LIN {X 0,Y 312.863,Z 418.471,A -85,B 0,C 180,E1 -15890.336,E2 -15890.336} C_VEL
LIN {X 0,Y 316.327,Z 432.665,A -85,B 0,C 180,E1 -15893.379,E2 -15893.379} C_VEL
LIN {X 0,Y 317.208,Z 437.346,A -85,B 0,C 180,E1 -15894.325,E2 -15894.325} C_VEL
LIN {X 0,Y 317.095,Z 438.182,A -85,B 0,C 180,E1 -15894.467,E2 -15894.467} C_VEL
LIN {X 0,Y 321.932,Z 475.252,A -85,B 0,C 180,E1 -15895.925,E2 -15895.925} C_VEL
LIN {X 0,Y 326.168,Z 512.092,A -85,B 0,C 180,E1 -15897.258,E2 -15897.258} C_VEL
LIN {X 0,Y 323.203,Z 607.757,A -85,B 0,C 180,E1 -15899.36,E2 -15899.36} C_VEL
LIN {X 0,Y 322.103,Z 623.409,A -85,B 0,C 180,E1 -15899.924,E2 -15899.924} C_VEL
LIN {X 0,Y 320.466,Z 638.482,A -85,B 0,C 180,E1 -15900.704,E2 -15900.704} C_VEL
LIN {X 0,Y 318.45,Z 652.595,A -85,B 0,C 180,E1 -15901.674,E2 -15901.674} C_VEL
LIN {X 0,Y 316.125,Z 666.999,A -85,B 0,C 180,E1 -15902.948,E2 -15902.948} C_VEL
LIN {X 0,Y 313.926,Z 680.599,A -85,B 0,C 180,E1 -15904.472,E2 -15904.472} C_VEL
LIN {X 0,Y 311.576,Z 693.378,A -85,B 0,C 180,E1 -15906.222,E2 -15906.222} C_VEL
LIN {X 0,Y 309.65,Z 704.13,A -85,B 0,C 180,E1 -15908.007,E2 -15908.007} C_VEL
LIN {X 0,Y 307.924,Z 714.131,A -85,B 0,C 180,E1 -15909.979,E2 -15909.979} C_VEL
LIN {X 0,Y 306.386,Z 723.981,A -85,B 0,C 180,E1 -15912.306,E2 -15912.306} C_VEL
LIN {X 0,Y 305.308,Z 732.423,A -85,B 0,C 180,E1 -15914.718,E2 -15914.718} C_VEL
LIN {X 0,Y 304.657,Z 739.918,A -85,B 0,C 180,E1 -15917.341,E2 -15917.341} C_VEL
LIN {X 0,Y 304.529,Z 746.052,A -85,B 0,C 180,E1 -15920.032,E2 -15920.032} C_VEL
LIN {X 0,Y 304.716,Z 750.636,A -85,B 0,C 180,E1 -15922.635,E2 -15922.635} C_VEL
LIN {X 0,Y 304.965,Z 753.357,A -85,B 0,C 180,E1 -15924.711,E2 -15924.711} C_VEL
LIN {X 0,Y 305.159,Z 755.666,A -85,B 0,C 180,E1 -15927.36,E2 -15927.36} C_VEL
LIN {X 0,Y 305.45,Z 756.378,A -85,B 0,C 180,E1 -15928.681,E2 -15928.681} C_VEL
LIN {X 0,Y 305.657,Z 756.769,A -85,B 0,C 180,E1 -15929.999,E2 -15929.999} C_VEL
LIN {X 0,Y 305.424,Z 756.792,A -85,B 0,C 180,E1 -15931.318,E2 -15931.318} C_VEL
LIN {X 0,Y 304.976,Z 755.908,A -85,B 0,C 180,E1 -15933.964,E2 -15933.964} C_VEL
LIN {X 0,Y 304.626,Z 753.778,A -85,B 0,C 180,E1 -15936.623,E2 -15936.623} C_VEL
LIN {X 0,Y 304.345,Z 750.421,A -85,B 0,C 180,E1 -15939.302,E2 -15939.302} C_VEL
LIN {X 0,Y 304.424,Z 745.812,A -85,B 0,C 180,E1 -15941.991,E2 -15941.991} C_VEL
LIN {X 0,Y 305.049,Z 739.867,A -85,B 0,C 180,E1 -15944.68,E2 -15944.68} C_VEL
LIN {X 0,Y 306.24,Z 732.446,A -85,B 0,C 180,E1 -15947.357,E2 -15947.357} C_VEL
LIN {X 0,Y 307.878,Z 724.631,A -85,B 0,C 180,E1 -15949.675,E2 -15949.675} C_VEL
LIN {X 0,Y 309.953,Z 715.588,A -85,B 0,C 180,E1 -15951.899,E2 -15951.899} C_VEL
LIN {X 0,Y 312.669,Z 704.202,A -85,B 0,C 180,E1 -15954.217,E2 -15954.217} C_VEL
LIN {X 0,Y 315.71,Z 691.846,A -85,B 0,C 180,E1 -15956.258,E2 -15956.258} C_VEL
LIN {X 0,Y 318.808,Z 679.206,A -85,B 0,C 180,E1 -15957.952,E2 -15957.952} C_VEL
LIN {X 0,Y 321.789,Z 665.625,A -85,B 0,C 180,E1 -15959.432,E2 -15959.432} C_VEL
LIN {X 0,Y 324.584,Z 652.223,A -85,B 0,C 180,E1 -15960.584,E2 -15960.584} C_VEL
LIN {X 0,Y 327.156,Z 637.542,A -85,B 0,C 180,E1 -15961.574,E2 -15961.574} C_VEL
LIN {X 0,Y 329.294,Z 622.301,A -85,B 0,C 180,E1 -15962.336,E2 -15962.336} C_VEL
LIN {X 0,Y 330.686,Z 606.3,A -85,B 0,C 180,E1 -15962.905,E2 -15962.905} C_VEL
LIN {X 0,Y 332.705,Z 555.604,A -85,B 0,C 180,E1 -15964.025,E2 -15964.025} C_VEL
LIN {X 0,Y 334.221,Z 512.744,A -85,B 0,C 180,E1 -15964.965,E2 -15964.965} C_VEL
LIN {X 0,Y 331.794,Z 490.509,A -85,B 0,C 180,E1 -15965.887,E2 -15965.887} C_VEL
LIN {X 0,Y 327.9,Z 463.19,A -85,B 0,C 180,E1 -15967.187,E2 -15967.187} C_VEL
LIN {X 0,Y 325.208,Z 447.828,A -85,B 0,C 180,E1 -15968.019,E2 -15968.019} C_VEL
LIN {X 0,Y 320.37,Z 437.85,A -85,B 0,C 180,E1 -15969.057,E2 -15969.057} C_VEL
LIN {X 0,Y 318.662,Z 434.062,A -85,B 0,C 180,E1 -15969.474,E2 -15969.474} C_VEL
LIN {X 0,Y 315.48,Z 422.569,A -85,B 0,C 180,E1 -15972.365,E2 -15972.365} C_VEL
LIN {X 0,Y 312.299,Z 412.488,A -85,B 0,C 180,E1 -15975.122,E2 -15975.122} C_VEL
LIN {X 0,Y 308.681,Z 402.063,A -85,B 0,C 180,E1 -15978.244,E2 -15978.244} C_VEL
LIN {X 0,Y 305.398,Z 393.062,A -85,B 0,C 180,E1 -15981.242,E2 -15981.242} C_VEL
LIN {X 0,Y 305.451,Z 393.062,A -85,B 0,C 180,E1 -15984.886,E2 -15984.886} C_VEL
LIN {X 0,Y 305.432,Z 393.066,A -85,B 0,C 180,E1 -15988.358,E2 -15988.358} C_VEL
LIN {X 0,Y 305.464,Z 393.064,A -85,B 0,C 180,E1 -15991.108,E2 -15991.108} C_VEL
LIN {X 0,Y 305.467,Z 393.064,A -85,B 0,C 180,E1 -15994.079,E2 -15994.079} C_VEL
LIN {X 0,Y 305.443,Z 393.06,A -85,B 0,C 180,E1 -15998.399,E2 -15998.399} C_VEL
LIN {X 0,Y 305.486,Z 393.06,A -85,B 0,C 180,E1 -16001.211,E2 -16001.211} C_VEL
LIN {X 0,Y 305.557,Z 393.047,A -85,B 0,C 180,E1 -16005.345,E2 -16005.345} C_VEL
LIN {X 0,Y 305.611,Z 393.035,A -85,B 0,C 180,E1 -16009.399,E2 -16009.399} C_VEL
LIN {X 0,Y 305.733,Z 393.029,A -85,B 0,C 180,E1 -16012.073,E2 -16012.073} C_VEL
LIN {X 0,Y 305.647,Z 393.034,A -85,B 0,C 180,E1 -16014.723,E2 -16014.723} C_VEL
LIN {X 0,Y 305.923,Z 393,A -85,B 0,C 180,E1 -16018.684,E2 -16018.684} C_VEL
LIN {X 0,Y 305.936,Z 392.992,A -85,B 0,C 180,E1 -16021.317,E2 -16021.317} C_VEL
LIN {X 0,Y 305.776,Z 392.982,A -85,B 0,C 180,E1 -16026.648,E2 -16026.648} C_VEL
LIN {X 0,Y 305.674,Z 393.019,A -85,B 0,C 180,E1 -16029.262,E2 -16029.262} C_VEL
LIN {X 0,Y 305.574,Z 393.019,A -85,B 0,C 180,E1 -16033.297,E2 -16033.297} C_VEL
LIN {X 0,Y 305.542,Z 393.033,A -85,B 0,C 180,E1 -16036.023,E2 -16036.023} C_VEL
LIN {X 0,Y 305.532,Z 393.035,A -85,B 0,C 180,E1 -16039.427,E2 -16039.427} C_VEL
LIN {X 0,Y 305.447,Z 393.055,A -85,B 0,C 180,E1 -16043.027,E2 -16043.027} C_VEL
LIN {X 0,Y 305.442,Z 393.042,A -85,B 0,C 180,E1 -16046.191,E2 -16046.191} C_VEL
LIN {X 0,Y 305.438,Z 393.064,A -85,B 0,C 180,E1 -16049.034,E2 -16049.034} C_VEL
LIN {X 0,Y 305.428,Z 393.046,A -85,B 0,C 180,E1 -16051.954,E2 -16051.954} C_VEL
LIN {X 0,Y 305.454,Z 393.062,A -85,B 0,C 180,E1 -16055.115,E2 -16055.115} C_VEL
LIN {X 0,Y 305.445,Z 393.061,A -85,B 0,C 180,E1 -16059.257,E2 -16059.257} C_VEL
LIN {X 0,Y 305.406,Z 393.058,A -85,B 0,C 180,E1 -16059.929,E2 -16059.929} C_VEL
LIN {X 0,Y 306.44,Z 395.935,A -85,B 0,C 180,E1 -16060.224,E2 -16060.224} C_VEL
LIN {X 0,Y 308.625,Z 398.473,A -85,B 0,C 180,E1 -16060.717,E2 -16060.717} C_VEL
LIN {X 0,Y 310.885,Z 401.914,A -85,B 0,C 180,E1 -16061.24,E2 -16061.24} C_VEL
LIN {X 0,Y 317.694,Z 411.904,A -85,B 0,C 180,E1 -16062.735,E2 -16062.735} C_VEL
LIN {X 0,Y 325.78,Z 424.373,A -85,B 0,C 180,E1 -16064.399,E2 -16064.399} C_VEL
LIN {X 0,Y 335.544,Z 441.537,A -85,B 0,C 180,E1 -16066.307,E2 -16066.307} C_VEL
LIN {X 0,Y 336.591,Z 443.642,A -85,B 0,C 180,E1 -16066.508,E2 -16066.508} C_VEL
LIN {X 0,Y 334.079,Z 511.752,A -85,B 0,C 180,E1 -16067.994,E2 -16067.994} C_VEL
LIN {X 0,Y 333.569,Z 531.567,A -85,B 0,C 180,E1 -16068.547,E2 -16068.547} C_VEL
LIN {X 0,Y 332.676,Z 546.26,A -85,B 0,C 180,E1 -16069.186,E2 -16069.186} C_VEL
LIN {X 0,Y 331.305,Z 560.291,A -85,B 0,C 180,E1 -16070.013,E2 -16070.013} C_VEL
LIN {X 0,Y 329.701,Z 573.58,A -85,B 0,C 180,E1 -16071.038,E2 -16071.038} C_VEL
LIN {X 0,Y 327.599,Z 586.902,A -85,B 0,C 180,E1 -16072.311,E2 -16072.311} C_VEL
LIN {X 0,Y 325.278,Z 599.133,A -85,B 0,C 180,E1 -16073.74,E2 -16073.74} C_VEL
LIN {X 0,Y 322.637,Z 611.425,A -85,B 0,C 180,E1 -16075.505,E2 -16075.505} C_VEL
LIN {X 0,Y 319.968,Z 622.521,A -85,B 0,C 180,E1 -16077.445,E2 -16077.445} C_VEL
LIN {X 0,Y 317.476,Z 631.8,A -85,B 0,C 180,E1 -16079.394,E2 -16079.394} C_VEL
LIN {X 0,Y 314.87,Z 640.813,A -85,B 0,C 180,E1 -16081.687,E2 -16081.687} C_VEL
LIN {X 0,Y 312.617,Z 648.371,A -85,B 0,C 180,E1 -16084.06,E2 -16084.06} C_VEL
LIN {X 0,Y 310.556,Z 655.033,A -85,B 0,C 180,E1 -16086.671,E2 -16086.671} C_VEL
LIN {X 0,Y 308.881,Z 660.345,A -85,B 0,C 180,E1 -16089.369,E2 -16089.369} C_VEL
LIN {X 0,Y 307.861,Z 663.372,A -85,B 0,C 180,E1 -16091.362,E2 -16091.362} C_VEL
LIN {X 0,Y 306.825,Z 666.441,A -85,B 0,C 180,E1 -16094.163,E2 -16094.163} C_VEL
LIN {X 0,Y 306.171,Z 668.127,A -85,B 0,C 180,E1 -16096.731,E2 -16096.731} C_VEL
LIN {X 0,Y 305.859,Z 668.735,A -85,B 0,C 180,E1 -16099.408,E2 -16099.408} C_VEL
LIN {X 0,Y 305.81,Z 668.241,A -85,B 0,C 180,E1 -16102.075,E2 -16102.075} C_VEL
LIN {X 0,Y 305.794,Z 666.691,A -85,B 0,C 180,E1 -16104.726,E2 -16104.726} C_VEL
LIN {X 0,Y 306.254,Z 663.988,A -85,B 0,C 180,E1 -16107.37,E2 -16107.37} C_VEL
LIN {X 0,Y 306.931,Z 660.111,A -85,B 0,C 180,E1 -16110.001,E2 -16110.001} C_VEL
LIN {X 0,Y 307.9,Z 654.945,A -85,B 0,C 180,E1 -16112.617,E2 -16112.617} C_VEL
LIN {X 0,Y 309.212,Z 648.379,A -85,B 0,C 180,E1 -16115.217,E2 -16115.217} C_VEL
LIN {X 0,Y 310.824,Z 640.233,A -85,B 0,C 180,E1 -16117.797,E2 -16117.797} C_VEL
LIN {X 0,Y 312.589,Z 631.524,A -85,B 0,C 180,E1 -16120.035,E2 -16120.035} C_VEL
LIN {X 0,Y 314.616,Z 621.082,A -85,B 0,C 180,E1 -16122.252,E2 -16122.252} C_VEL
LIN {X 0,Y 316.523,Z 610.337,A -85,B 0,C 180,E1 -16124.137,E2 -16124.137} C_VEL
LIN {X 0,Y 318.251,Z 598.642,A -85,B 0,C 180,E1 -16125.86,E2 -16125.86} C_VEL
LIN {X 0,Y 320.198,Z 585.754,A -85,B 0,C 180,E1 -16127.401,E2 -16127.401} C_VEL
LIN {X 0,Y 321.779,Z 573.192,A -85,B 0,C 180,E1 -16128.628,E2 -16128.628} C_VEL
LIN {X 0,Y 323.227,Z 559.555,A -85,B 0,C 180,E1 -16129.695,E2 -16129.695} C_VEL
LIN {X 0,Y 324.421,Z 544.22,A -85,B 0,C 180,E1 -16130.616,E2 -16130.616} C_VEL
LIN {X 0,Y 325.083,Z 529.118,A -85,B 0,C 180,E1 -16131.27,E2 -16131.27} C_VEL
LIN {X 0,Y 325.477,Z 509.141,A -85,B 0,C 180,E1 -16131.807,E2 -16131.807} C_VEL
LIN {X 0,Y 327.521,Z 435.989,A -85,B 0,C 180,E1 -16133.421,E2 -16133.421} C_VEL
LIN {X 0,Y 319.152,Z 418.636,A -85,B 0,C 180,E1 -16134.742,E2 -16134.742} C_VEL
LIN {X 0,Y 309.104,Z 400.268,A -85,B 0,C 180,E1 -16136.381,E2 -16136.381} C_VEL
LIN {X 0,Y 306.929,Z 396.598,A -85,B 0,C 180,E1 -16136.745,E2 -16136.745} C_VEL
LIN {X 0,Y 305.623,Z 394.015,A -85,B 0,C 180,E1 -16136.977,E2 -16136.977} C_VEL
LIN {X 0,Y 305.436,Z 393.065,A -85,B 0,C 180,E1 -16137.068,E2 -16137.068} C_VEL
LIN {X 0,Y 305.409,Z 393.05,A -85,B 0,C 180,E1 -16140.706,E2 -16140.706} C_VEL
LIN {X 0,Y 305.465,Z 393.056,A -85,B 0,C 180,E1 -16144.078,E2 -16144.078} C_VEL
LIN {X 0,Y 305.459,Z 393.057,A -85,B 0,C 180,E1 -16146.431,E2 -16146.431} C_VEL
LIN {X 0,Y 304.758,Z 393.147,A -85,B 0,C 180,E1 -16147.53,E2 -16147.53} C_VEL
LIN {X 0,Y 301.851,Z 393.505,A -85,B 0,C 180,E1 -16149.318,E2 -16149.318} C_VEL
LIN {X 0,Y 299.414,Z 393.808,A -85,B 0,C 180,E1 -16150.769,E2 -16150.769} C_VEL
LIN {X 0,Y 298.389,Z 393.941,A -85,B 0,C 180,E1 -16151.893,E2 -16151.893} C_VEL
LIN {X 0,Y 298.316,Z 393.942,A -85,B 0,C 180,E1 -16152.274,E2 -16152.274} C_VEL
LIN {X 0,Y 298.354,Z 393.945,A -85,B 0,C 180,E1 -16155.034,E2 -16155.034} C_VEL
LIN {X 0,Y 298.345,Z 393.946,A -85,B 0,C 180,E1 -16158.921,E2 -16158.921} C_VEL
LIN {X 0,Y 298.423,Z 393.937,A -85,B 0,C 180,E1 -16163.197,E2 -16163.197} C_VEL
LIN {X 0,Y 298.404,Z 393.932,A -85,B 0,C 180,E1 -16165.58,E2 -16165.58} C_VEL
LIN {X 0,Y 298.366,Z 393.946,A -85,B 0,C 180,E1 -16168.787,E2 -16168.787} C_VEL
LIN {X 0,Y 298.392,Z 393.937,A -85,B 0,C 180,E1 -16171.897,E2 -16171.897} C_VEL
LIN {X 0,Y 298.434,Z 393.932,A -85,B 0,C 180,E1 -16174.919,E2 -16174.919} C_VEL
LIN {X 0,Y 298.396,Z 393.941,A -85,B 0,C 180,E1 -16177.861,E2 -16177.861} C_VEL
LIN {X 0,Y 298.459,Z 393.923,A -85,B 0,C 180,E1 -16180.751,E2 -16180.751} C_VEL
LIN {X 0,Y 298.582,Z 393.915,A -85,B 0,C 180,E1 -16184.994,E2 -16184.994} C_VEL
LIN {X 0,Y 298.576,Z 393.866,A -85,B 0,C 180,E1 -16189.146,E2 -16189.146} C_VEL
LIN {X 0,Y 298.678,Z 393.883,A -85,B 0,C 180,E1 -16191.883,E2 -16191.883} C_VEL
LIN {X 0,Y 298.616,Z 393.912,A -85,B 0,C 180,E1 -16194.598,E2 -16194.598} C_VEL
LIN {X 0,Y 298.9,Z 393.865,A -85,B 0,C 180,E1 -16198.652,E2 -16198.652} C_VEL
LIN {X 0,Y 298.896,Z 393.879,A -85,B 0,C 180,E1 -16201.347,E2 -16201.347} C_VEL
LIN {X 0,Y 298.723,Z 393.898,A -85,B 0,C 180,E1 -16206.755,E2 -16206.755} C_VEL
LIN {X 0,Y 298.619,Z 393.9,A -85,B 0,C 180,E1 -16209.482,E2 -16209.482} C_VEL
LIN {X 0,Y 298.509,Z 393.918,A -85,B 0,C 180,E1 -16213.617,E2 -16213.617} C_VEL
LIN {X 0,Y 298.43,Z 393.936,A -85,B 0,C 180,E1 -16216.415,E2 -16216.415} C_VEL
LIN {X 0,Y 298.425,Z 393.931,A -85,B 0,C 180,E1 -16219.61,E2 -16219.61} C_VEL
LIN {X 0,Y 298.382,Z 393.937,A -85,B 0,C 180,E1 -16223.604,E2 -16223.604} C_VEL
LIN {X 0,Y 298.395,Z 393.935,A -85,B 0,C 180,E1 -16226.583,E2 -16226.583} C_VEL
LIN {X 0,Y 298.352,Z 393.943,A -85,B 0,C 180,E1 -16229.648,E2 -16229.648} C_VEL
LIN {X 0,Y 298.388,Z 393.93,A -85,B 0,C 180,E1 -16232.801,E2 -16232.801} C_VEL
LIN {X 0,Y 298.399,Z 393.945,A -85,B 0,C 180,E1 -16236.072,E2 -16236.072} C_VEL
LIN {X 0,Y 298.369,Z 393.934,A -85,B 0,C 180,E1 -16239.492,E2 -16239.492} C_VEL
LIN {X 0,Y 298.386,Z 394.058,A -85,B 0,C 180,E1 -16243.545,E2 -16243.545} C_VEL
LIN {X 0,Y 302.653,Z 407.836,A -85,B 0,C 180,E1 -16247.062,E2 -16247.062} C_VEL
LIN {X 0,Y 306.461,Z 421.574,A -85,B 0,C 180,E1 -16250.292,E2 -16250.292} C_VEL
LIN {X 0,Y 310.134,Z 436.942,A -85,B 0,C 180,E1 -16253.645,E2 -16253.645} C_VEL
LIN {X 0,Y 311.139,Z 440.411,A -85,B 0,C 180,E1 -16253.863,E2 -16253.863} C_VEL
LIN {X 0,Y 314.949,Z 469.814,A -85,B 0,C 180,E1 -16255.057,E2 -16255.057} C_VEL
LIN {X 0,Y 319.897,Z 512.328,A -85,B 0,C 180,E1 -16256.656,E2 -16256.656} C_VEL
LIN {X 0,Y 316.891,Z 606.888,A -85,B 0,C 180,E1 -16258.775,E2 -16258.775} C_VEL
LIN {X 0,Y 315.747,Z 622.48,A -85,B 0,C 180,E1 -16259.346,E2 -16259.346} C_VEL
LIN {X 0,Y 314.064,Z 637.53,A -85,B 0,C 180,E1 -16260.139,E2 -16260.139} C_VEL
LIN {X 0,Y 311.856,Z 652.629,A -85,B 0,C 180,E1 -16261.203,E2 -16261.203} C_VEL
LIN {X 0,Y 309.362,Z 667.426,A -85,B 0,C 180,E1 -16262.565,E2 -16262.565} C_VEL
LIN {X 0,Y 307.204,Z 680.266,A -85,B 0,C 180,E1 -16264.054,E2 -16264.054} C_VEL
LIN {X 0,Y 304.762,Z 692.926,A -85,B 0,C 180,E1 -16265.838,E2 -16265.838} C_VEL
LIN {X 0,Y 302.622,Z 704.52,A -85,B 0,C 180,E1 -16267.828,E2 -16267.828} C_VEL
LIN {X 0,Y 300.597,Z 715.806,A -85,B 0,C 180,E1 -16270.183,E2 -16270.183} C_VEL
LIN {X 0,Y 299.128,Z 725.224,A -85,B 0,C 180,E1 -16272.569,E2 -16272.569} C_VEL
LIN {X 0,Y 298.136,Z 733.542,A -85,B 0,C 180,E1 -16275.127,E2 -16275.127} C_VEL
LIN {X 0,Y 297.529,Z 740.406,A -85,B 0,C 180,E1 -16277.726,E2 -16277.726} C_VEL
LIN {X 0,Y 297.489,Z 746.205,A -85,B 0,C 180,E1 -16280.481,E2 -16280.481} C_VEL
LIN {X 0,Y 297.699,Z 750.571,A -85,B 0,C 180,E1 -16283.221,E2 -16283.221} C_VEL
LIN {X 0,Y 297.901,Z 752.252,A -85,B 0,C 180,E1 -16284.585,E2 -16284.585} C_VEL
LIN {X 0,Y 298.119,Z 754.604,A -85,B 0,C 180,E1 -16287.297,E2 -16287.297} C_VEL
LIN {X 0,Y 298.419,Z 755.335,A -85,B 0,C 180,E1 -16288.65,E2 -16288.65} C_VEL
LIN {X 0,Y 298.639,Z 755.746,A -85,B 0,C 180,E1 -16289.999,E2 -16289.999} C_VEL
LIN {X 0,Y 298.389,Z 755.783,A -85,B 0,C 180,E1 -16291.349,E2 -16291.349} C_VEL
LIN {X 0,Y 297.928,Z 754.911,A -85,B 0,C 180,E1 -16294.058,E2 -16294.058} C_VEL
LIN {X 0,Y 297.555,Z 752.809,A -85,B 0,C 180,E1 -16296.782,E2 -16296.782} C_VEL
LIN {X 0,Y 297.25,Z 749.478,A -85,B 0,C 180,E1 -16299.526,E2 -16299.526} C_VEL
LIN {X 0,Y 297.37,Z 744.904,A -85,B 0,C 180,E1 -16302.28,E2 -16302.28} C_VEL
LIN {X 0,Y 298.086,Z 739.004,A -85,B 0,C 180,E1 -16305.03,E2 -16305.03} C_VEL
LIN {X 0,Y 299.349,Z 731.63,A -85,B 0,C 180,E1 -16307.77,E2 -16307.77} C_VEL
LIN {X 0,Y 301.425,Z 722.606,A -85,B 0,C 180,E1 -16310.47,E2 -16310.47} C_VEL
LIN {X 0,Y 303.713,Z 713.119,A -85,B 0,C 180,E1 -16312.804,E2 -16312.804} C_VEL
LIN {X 0,Y 306.137,Z 703.54,A -85,B 0,C 180,E1 -16314.768,E2 -16314.768} C_VEL
LIN {X 0,Y 309.036,Z 692.279,A -85,B 0,C 180,E1 -16316.688,E2 -16316.688} C_VEL
LIN {X 0,Y 312.27,Z 679.69,A -85,B 0,C 180,E1 -16318.443,E2 -16318.443} C_VEL
LIN {X 0,Y 315.274,Z 666.723,A -85,B 0,C 180,E1 -16319.918,E2 -16319.918} C_VEL
LIN {X 0,Y 318.094,Z 653.792,A -85,B 0,C 180,E1 -16321.093,E2 -16321.093} C_VEL
LIN {X 0,Y 320.758,Z 639.838,A -85,B 0,C 180,E1 -16322.094,E2 -16322.094} C_VEL
LIN {X 0,Y 323.133,Z 624.249,A -85,B 0,C 180,E1 -16322.937,E2 -16322.937} C_VEL
LIN {X 0,Y 324.674,Z 608.626,A -85,B 0,C 180,E1 -16323.548,E2 -16323.548} C_VEL
LIN {X 0,Y 325.676,Z 590.836,A -85,B 0,C 180,E1 -16323.988,E2 -16323.988} C_VEL
LIN {X 0,Y 328.594,Z 513.907,A -85,B 0,C 180,E1 -16325.687,E2 -16325.687} C_VEL
LIN {X 0,Y 326.244,Z 491.87,A -85,B 0,C 180,E1 -16326.624,E2 -16326.624} C_VEL
LIN {X 0,Y 322.613,Z 465.718,A -85,B 0,C 180,E1 -16327.898,E2 -16327.898} C_VEL
LIN {X 0,Y 320.055,Z 450.931,A -85,B 0,C 180,E1 -16328.722,E2 -16328.722} C_VEL
LIN {X 0,Y 313.785,Z 437.959,A -85,B 0,C 180,E1 -16330.131,E2 -16330.131} C_VEL
LIN {X 0,Y 311.211,Z 432.729,A -85,B 0,C 180,E1 -16330.737,E2 -16330.737} C_VEL
LIN {X 0,Y 308.051,Z 421.743,A -85,B 0,C 180,E1 -16333.65,E2 -16333.65} C_VEL
LIN {X 0,Y 304.231,Z 410.145,A -85,B 0,C 180,E1 -16337.041,E2 -16337.041} C_VEL
LIN {X 0,Y 300.893,Z 400.885,A -85,B 0,C 180,E1 -16340.036,E2 -16340.036} C_VEL
LIN {X 0,Y 298.364,Z 393.947,A -85,B 0,C 180,E1 -16342.505,E2 -16342.505} C_VEL
LIN {X 0,Y 298.398,Z 393.94,A -85,B 0,C 180,E1 -16345.58,E2 -16345.58} C_VEL
LIN {X 0,Y 298.367,Z 393.942,A -85,B 0,C 180,E1 -16348.788,E2 -16348.788} C_VEL
LIN {X 0,Y 298.398,Z 393.939,A -85,B 0,C 180,E1 -16351.898,E2 -16351.898} C_VEL
LIN {X 0,Y 298.401,Z 393.94,A -85,B 0,C 180,E1 -16354.917,E2 -16354.917} C_VEL
LIN {X 0,Y 298.378,Z 393.947,A -85,B 0,C 180,E1 -16357.861,E2 -16357.861} C_VEL
LIN {X 0,Y 298.438,Z 393.94,A -85,B 0,C 180,E1 -16360.75,E2 -16360.75} C_VEL
LIN {X 0,Y 298.499,Z 393.928,A -85,B 0,C 180,E1 -16364.99,E2 -16364.99} C_VEL
LIN {X 0,Y 298.569,Z 393.914,A -85,B 0,C 180,E1 -16369.146,E2 -16369.146} C_VEL
LIN {X 0,Y 298.685,Z 393.906,A -85,B 0,C 180,E1 -16371.884,E2 -16371.884} C_VEL
LIN {X 0,Y 298.616,Z 393.908,A -85,B 0,C 180,E1 -16374.598,E2 -16374.598} C_VEL
LIN {X 0,Y 298.891,Z 393.876,A -85,B 0,C 180,E1 -16378.653,E2 -16378.653} C_VEL
LIN {X 0,Y 298.902,Z 393.868,A -85,B 0,C 180,E1 -16381.348,E2 -16381.348} C_VEL
LIN {X 0,Y 298.728,Z 393.858,A -85,B 0,C 180,E1 -16386.756,E2 -16386.756} C_VEL
LIN {X 0,Y 298.572,Z 393.92,A -85,B 0,C 180,E1 -16390.855,E2 -16390.855} C_VEL
LIN {X 0,Y 298.538,Z 393.892,A -85,B 0,C 180,E1 -16395.168,E2 -16395.168} C_VEL
LIN {X 0,Y 298.494,Z 393.913,A -85,B 0,C 180,E1 -16399.247,E2 -16399.247} C_VEL
LIN {X 0,Y 298.379,Z 393.943,A -85,B 0,C 180,E1 -16403.605,E2 -16403.605} C_VEL
LIN {X 0,Y 298.394,Z 393.917,A -85,B 0,C 180,E1 -16406.584,E2 -16406.584} C_VEL
LIN {X 0,Y 298.384,Z 393.946,A -85,B 0,C 180,E1 -16409.645,E2 -16409.645} C_VEL
LIN {X 0,Y 298.385,Z 393.927,A -85,B 0,C 180,E1 -16412.802,E2 -16412.802} C_VEL
LIN {X 0,Y 298.397,Z 393.929,A -85,B 0,C 180,E1 -16416.073,E2 -16416.073} C_VEL
LIN {X 0,Y 298.4,Z 393.994,A -85,B 0,C 180,E1 -16418.563,E2 -16418.563} C_VEL
LIN {X 0,Y 299.334,Z 396.675,A -85,B 0,C 180,E1 -16418.849,E2 -16418.849} C_VEL
LIN {X 0,Y 301.792,Z 399.575,A -85,B 0,C 180,E1 -16419.444,E2 -16419.444} C_VEL
LIN {X 0,Y 303.792,Z 402.692,A -85,B 0,C 180,E1 -16419.94,E2 -16419.94} C_VEL
LIN {X 0,Y 305.15,Z 404.437,A -85,B 0,C 180,E1 -16420.258,E2 -16420.258} C_VEL
LIN {X 0,Y 313.61,Z 416.842,A -85,B 0,C 180,E1 -16422.191,E2 -16422.191} C_VEL
LIN {X 0,Y 322.184,Z 430.425,A -85,B 0,C 180,E1 -16424.015,E2 -16424.015} C_VEL
LIN {X 0,Y 330.885,Z 445.856,A -85,B 0,C 180,E1 -16425.766,E2 -16425.766} C_VEL
LIN {X 0,Y 329.577,Z 481.898,A -85,B 0,C 180,E1 -16426.576,E2 -16426.576} C_VEL
LIN {X 0,Y 328.409,Z 515.364,A -85,B 0,C 180,E1 -16427.332,E2 -16427.332} C_VEL
LIN {X 0,Y 327.87,Z 533.034,A -85,B 0,C 180,E1 -16427.843,E2 -16427.843} C_VEL
LIN {X 0,Y 326.971,Z 547.313,A -85,B 0,C 180,E1 -16428.478,E2 -16428.478} C_VEL
LIN {X 0,Y 325.499,Z 561.584,A -85,B 0,C 180,E1 -16429.333,E2 -16429.333} C_VEL
LIN {X 0,Y 323.795,Z 575.005,A -85,B 0,C 180,E1 -16430.39,E2 -16430.39} C_VEL
LIN {X 0,Y 321.685,Z 587.835,A -85,B 0,C 180,E1 -16431.635,E2 -16431.635} C_VEL
LIN {X 0,Y 319.211,Z 600.43,A -85,B 0,C 180,E1 -16433.135,E2 -16433.135} C_VEL
LIN {X 0,Y 316.69,Z 611.66,A -85,B 0,C 180,E1 -16434.762,E2 -16434.762} C_VEL
LIN {X 0,Y 313.865,Z 622.893,A -85,B 0,C 180,E1 -16436.731,E2 -16436.731} C_VEL
LIN {X 0,Y 311.247,Z 632.251,A -85,B 0,C 180,E1 -16438.713,E2 -16438.713} C_VEL
LIN {X 0,Y 308.525,Z 641.36,A -85,B 0,C 180,E1 -16441.05,E2 -16441.05} C_VEL
LIN {X 0,Y 306.047,Z 649.338,A -85,B 0,C 180,E1 -16443.585,E2 -16443.585} C_VEL
LIN {X 0,Y 303.931,Z 655.748,A -85,B 0,C 180,E1 -16446.131,E2 -16446.131} C_VEL
LIN {X 0,Y 302.094,Z 661.255,A -85,B 0,C 180,E1 -16448.956,E2 -16448.956} C_VEL
LIN {X 0,Y 301.05,Z 664.229,A -85,B 0,C 180,E1 -16450.925,E2 -16450.925} C_VEL
LIN {X 0,Y 299.853,Z 667.481,A -85,B 0,C 180,E1 -16453.94,E2 -16453.94} C_VEL
LIN {X 0,Y 299.202,Z 669.078,A -85,B 0,C 180,E1 -16456.416,E2 -16456.416} C_VEL
LIN {X 0,Y 298.866,Z 669.742,A -85,B 0,C 180,E1 -16459.157,E2 -16459.157} C_VEL
LIN {X 0,Y 298.783,Z 669.309,A -85,B 0,C 180,E1 -16461.887,E2 -16461.887} C_VEL
LIN {X 0,Y 298.768,Z 667.815,A -85,B 0,C 180,E1 -16464.602,E2 -16464.602} C_VEL
LIN {X 0,Y 299.207,Z 665.177,A -85,B 0,C 180,E1 -16467.308,E2 -16467.308} C_VEL
LIN {X 0,Y 299.916,Z 661.335,A -85,B 0,C 180,E1 -16470.001,E2 -16470.001} C_VEL
LIN {X 0,Y 300.901,Z 656.228,A -85,B 0,C 180,E1 -16472.678,E2 -16472.678} C_VEL
LIN {X 0,Y 302.246,Z 649.734,A -85,B 0,C 180,E1 -16475.337,E2 -16475.337} C_VEL
LIN {X 0,Y 303.914,Z 641.668,A -85,B 0,C 180,E1 -16477.976,E2 -16477.976} C_VEL
LIN {X 0,Y 305.741,Z 633.047,A -85,B 0,C 180,E1 -16480.262,E2 -16480.262} C_VEL
LIN {X 0,Y 307.808,Z 622.714,A -85,B 0,C 180,E1 -16482.528,E2 -16482.528} C_VEL
LIN {X 0,Y 309.791,Z 612.09,A -85,B 0,C 180,E1 -16484.451,E2 -16484.451} C_VEL
LIN {X 0,Y 311.602,Z 600.541,A -85,B 0,C 180,E1 -16486.207,E2 -16486.207} C_VEL
LIN {X 0,Y 313.607,Z 587.848,A -85,B 0,C 180,E1 -16487.779,E2 -16487.779} C_VEL
LIN {X 0,Y 315.221,Z 575.553,A -85,B 0,C 180,E1 -16489.03,E2 -16489.03} C_VEL
LIN {X 0,Y 316.819,Z 561.197,A -85,B 0,C 180,E1 -16490.195,E2 -16490.195} C_VEL
LIN {X 0,Y 318.085,Z 546.052,A -85,B 0,C 180,E1 -16491.132,E2 -16491.132} C_VEL
LIN {X 0,Y 318.818,Z 531.613,A -85,B 0,C 180,E1 -16491.784,E2 -16491.784} C_VEL
LIN {X 0,Y 319.173,Z 514.301,A -85,B 0,C 180,E1 -16492.291,E2 -16492.291} C_VEL
LIN {X 0,Y 321.375,Z 438.213,A -85,B 0,C 180,E1 -16494,E2 -16494} C_VEL
LIN {X 0,Y 313.916,Z 422.594,A -85,B 0,C 180,E1 -16495.221,E2 -16495.221} C_VEL
LIN {X 0,Y 304.148,Z 404.641,A -85,B 0,C 180,E1 -16496.865,E2 -16496.865} C_VEL
LIN {X 0,Y 299.895,Z 397.475,A -85,B 0,C 180,E1 -16497.605,E2 -16497.605} C_VEL
LIN {X 0,Y 298.617,Z 395.068,A -85,B 0,C 180,E1 -16497.84,E2 -16497.84} C_VEL
LIN {X 0,Y 298.384,Z 393.946,A -85,B 0,C 180,E1 -16497.944,E2 -16497.944} C_VEL
LIN {X 0,Y 298.388,Z 393.944,A -85,B 0,C 180,E1 -16502.013,E2 -16502.013} C_VEL
LIN {X 0,Y 298.429,Z 393.934,A -85,B 0,C 180,E1 -16504.487,E2 -16504.487} C_VEL
LIN {X 0,Y 298.391,Z 393.941,A -85,B 0,C 180,E1 -16507.761,E2 -16507.761} C_VEL
LIN {X 0,Y 298.335,Z 393.947,A -85,B 0,C 180,E1 -16511.269,E2 -16511.269} C_VEL
LIN {X 0,Y 298.316,Z 393.942,A -85,B 0,C 180,E1 -16512.274,E2 -16512.274} C_VEL
LIN {X 0,Y 297.669,Z 394.027,A -85,B 0,C 180,E1 -16513.402,E2 -16513.402} C_VEL
LIN {X 0,Y 294.803,Z 394.389,A -85,B 0,C 180,E1 -16515.237,E2 -16515.237} C_VEL
LIN {X 0,Y 292.374,Z 394.687,A -85,B 0,C 180,E1 -16516.727,E2 -16516.727} C_VEL
LIN {X 0,Y 291.355,Z 394.811,A -85,B 0,C 180,E1 -16517.881,E2 -16517.881} C_VEL
LIN {X 0,Y 291.286,Z 394.821,A -85,B 0,C 180,E1 -16518.272,E2 -16518.272} C_VEL
LIN {X 0,Y 291.303,Z 394.818,A -85,B 0,C 180,E1 -16521.15,E2 -16521.15} C_VEL
LIN {X 0,Y 291.352,Z 394.82,A -85,B 0,C 180,E1 -16524.624,E2 -16524.624} C_VEL
LIN {X 0,Y 291.36,Z 394.818,A -85,B 0,C 180,E1 -16527.949,E2 -16527.949} C_VEL
LIN {X 0,Y 291.31,Z 394.815,A -85,B 0,C 180,E1 -16531.15,E2 -16531.15} C_VEL
LIN {X 0,Y 291.354,Z 394.816,A -85,B 0,C 180,E1 -16534.266,E2 -16534.266} C_VEL
LIN {X 0,Y 291.36,Z 394.812,A -85,B 0,C 180,E1 -16537.297,E2 -16537.297} C_VEL
LIN {X 0,Y 291.387,Z 394.806,A -85,B 0,C 180,E1 -16540.265,E2 -16540.265} C_VEL
LIN {X 0,Y 291.494,Z 394.799,A -85,B 0,C 180,E1 -16544.665,E2 -16544.665} C_VEL
LIN {X 0,Y 291.522,Z 394.744,A -85,B 0,C 180,E1 -16548.88,E2 -16548.88} C_VEL
LIN {X 0,Y 291.624,Z 394.758,A -85,B 0,C 180,E1 -16551.686,E2 -16551.686} C_VEL
LIN {X 0,Y 291.587,Z 394.787,A -85,B 0,C 180,E1 -16554.467,E2 -16554.467} C_VEL
LIN {X 0,Y 291.866,Z 394.741,A -85,B 0,C 180,E1 -16558.62,E2 -16558.62} C_VEL
LIN {X 0,Y 291.864,Z 394.754,A -85,B 0,C 180,E1 -16561.379,E2 -16561.379} C_VEL
LIN {X 0,Y 291.676,Z 394.776,A -85,B 0,C 180,E1 -16566.919,E2 -16566.919} C_VEL
LIN {X 0,Y 291.562,Z 394.78,A -85,B 0,C 180,E1 -16569.714,E2 -16569.714} C_VEL
LIN {X 0,Y 291.47,Z 394.793,A -85,B 0,C 180,E1 -16573.952,E2 -16573.952} C_VEL
LIN {X 0,Y 291.367,Z 394.808,A -85,B 0,C 180,E1 -16578.274,E2 -16578.274} C_VEL
LIN {X 0,Y 291.335,Z 394.822,A -85,B 0,C 180,E1 -16581.214,E2 -16581.214} C_VEL
LIN {X 0,Y 291.327,Z 394.822,A -85,B 0,C 180,E1 -16584.211,E2 -16584.211} C_VEL
LIN {X 0,Y 291.323,Z 394.818,A -85,B 0,C 180,E1 -16587.281,E2 -16587.281} C_VEL
LIN {X 0,Y 291.297,Z 394.826,A -85,B 0,C 180,E1 -16590.441,E2 -16590.441} C_VEL
LIN {X 0,Y 291.338,Z 394.802,A -85,B 0,C 180,E1 -16593.699,E2 -16593.699} C_VEL
LIN {X 0,Y 291.343,Z 394.814,A -85,B 0,C 180,E1 -16597.246,E2 -16597.246} C_VEL
LIN {X 0,Y 291.295,Z 394.827,A -85,B 0,C 180,E1 -16600.648,E2 -16600.648} C_VEL
LIN {X 0,Y 291.325,Z 394.997,A -85,B 0,C 180,E1 -16602.749,E2 -16602.749} C_VEL
LIN {X 0,Y 295.753,Z 408.86,A -85,B 0,C 180,E1 -16606.44,E2 -16606.44} C_VEL
LIN {X 0,Y 299.444,Z 422.341,A -85,B 0,C 180,E1 -16609.71,E2 -16609.71} C_VEL
LIN {X 0,Y 302.691,Z 435.822,A -85,B 0,C 180,E1 -16612.747,E2 -16612.747} C_VEL
LIN {X 0,Y 305.189,Z 442.17,A -85,B 0,C 180,E1 -16613.221,E2 -16613.221} C_VEL
LIN {X 0,Y 308.86,Z 470.834,A -85,B 0,C 180,E1 -16614.418,E2 -16614.418} C_VEL
LIN {X 0,Y 313.705,Z 513.834,A -85,B 0,C 180,E1 -16616.067,E2 -16616.067} C_VEL
LIN {X 0,Y 310.624,Z 606.021,A -85,B 0,C 180,E1 -16618.167,E2 -16618.167} C_VEL
LIN {X 0,Y 309.433,Z 621.554,A -85,B 0,C 180,E1 -16618.746,E2 -16618.746} C_VEL
LIN {X 0,Y 307.734,Z 636.592,A -85,B 0,C 180,E1 -16619.555,E2 -16619.555} C_VEL
LIN {X 0,Y 305.611,Z 650.675,A -85,B 0,C 180,E1 -16620.558,E2 -16620.558} C_VEL
LIN {X 0,Y 303.307,Z 663.911,A -85,B 0,C 180,E1 -16621.76,E2 -16621.76} C_VEL
LIN {X 0,Y 300.968,Z 677.3,A -85,B 0,C 180,E1 -16623.288,E2 -16623.288} C_VEL
LIN {X 0,Y 298.612,Z 689.188,A -85,B 0,C 180,E1 -16624.936,E2 -16624.936} C_VEL
LIN {X 0,Y 296.253,Z 701.207,A -85,B 0,C 180,E1 -16626.957,E2 -16626.957} C_VEL
LIN {X 0,Y 294.33,Z 711.35,A -85,B 0,C 180,E1 -16629.012,E2 -16629.012} C_VEL
LIN {X 0,Y 292.642,Z 721.332,A -85,B 0,C 180,E1 -16631.445,E2 -16631.445} C_VEL
LIN {X 0,Y 291.376,Z 729.66,A -85,B 0,C 180,E1 -16633.896,E2 -16633.896} C_VEL
LIN {X 0,Y 290.783,Z 735.701,A -85,B 0,C 180,E1 -16636.013,E2 -16636.013} C_VEL
LIN {X 0,Y 290.377,Z 742.29,A -85,B 0,C 180,E1 -16638.835,E2 -16638.835} C_VEL
LIN {X 0,Y 290.503,Z 747.411,A -85,B 0,C 180,E1 -16641.653,E2 -16641.653} C_VEL
LIN {X 0,Y 290.839,Z 751.147,A -85,B 0,C 180,E1 -16644.453,E2 -16644.453} C_VEL
LIN {X 0,Y 291.078,Z 753.542,A -85,B 0,C 180,E1 -16647.232,E2 -16647.232} C_VEL
LIN {X 0,Y 291.387,Z 754.293,A -85,B 0,C 180,E1 -16648.617,E2 -16648.617} C_VEL
LIN {X 0,Y 291.62,Z 754.722,A -85,B 0,C 180,E1 -16649.999,E2 -16649.999} C_VEL
LIN {X 0,Y 291.354,Z 754.774,A -85,B 0,C 180,E1 -16651.382,E2 -16651.382} C_VEL
LIN {X 0,Y 290.882,Z 753.915,A -85,B 0,C 180,E1 -16654.156,E2 -16654.156} C_VEL
LIN {X 0,Y 290.458,Z 751.835,A -85,B 0,C 180,E1 -16656.948,E2 -16656.948} C_VEL
LIN {X 0,Y 290.177,Z 748.539,A -85,B 0,C 180,E1 -16659.76,E2 -16659.76} C_VEL
LIN {X 0,Y 290.333,Z 744.002,A -85,B 0,C 180,E1 -16662.582,E2 -16662.582} C_VEL
LIN {X 0,Y 291.11,Z 738.144,A -85,B 0,C 180,E1 -16665.399,E2 -16665.399} C_VEL
LIN {X 0,Y 292.471,Z 730.816,A -85,B 0,C 180,E1 -16668.202,E2 -16668.202} C_VEL
LIN {X 0,Y 294.688,Z 721.847,A -85,B 0,C 180,E1 -16670.96,E2 -16670.96} C_VEL
LIN {X 0,Y 297.065,Z 712.417,A -85,B 0,C 180,E1 -16673.344,E2 -16673.344} C_VEL
LIN {X 0,Y 300.073,Z 701.149,A -85,B 0,C 180,E1 -16675.675,E2 -16675.675} C_VEL
LIN {X 0,Y 303.277,Z 689.695,A -85,B 0,C 180,E1 -16677.61,E2 -16677.61} C_VEL
LIN {X 0,Y 306.676,Z 676.394,A -85,B 0,C 180,E1 -16679.445,E2 -16679.445} C_VEL
LIN {X 0,Y 309.816,Z 663.472,A -85,B 0,C 180,E1 -16680.878,E2 -16680.878} C_VEL
LIN {X 0,Y 312.811,Z 650.071,A -85,B 0,C 180,E1 -16682.057,E2 -16682.057} C_VEL
LIN {X 0,Y 315.584,Z 635.386,A -85,B 0,C 180,E1 -16683.065,E2 -16683.065} C_VEL
LIN {X 0,Y 317.835,Z 620.134,A -85,B 0,C 180,E1 -16683.843,E2 -16683.843} C_VEL
LIN {X 0,Y 319.378,Z 604.094,A -85,B 0,C 180,E1 -16684.419,E2 -16684.419} C_VEL
LIN {X 0,Y 323.006,Z 515.015,A -85,B 0,C 180,E1 -16686.438,E2 -16686.438} C_VEL
LIN {X 0,Y 320.941,Z 494.628,A -85,B 0,C 180,E1 -16687.319,E2 -16687.319} C_VEL
LIN {X 0,Y 317.286,Z 467.648,A -85,B 0,C 180,E1 -16688.666,E2 -16688.666} C_VEL
LIN {X 0,Y 314.949,Z 453.902,A -85,B 0,C 180,E1 -16689.453,E2 -16689.453} C_VEL
LIN {X 0,Y 308.402,Z 440.572,A -85,B 0,C 180,E1 -16690.98,E2 -16690.98} C_VEL
LIN {X 0,Y 305.347,Z 434.75,A -85,B 0,C 180,E1 -16691.717,E2 -16691.717} C_VEL
LIN {X 0,Y 303.588,Z 430.961,A -85,B 0,C 180,E1 -16692.201,E2 -16692.201} C_VEL
LIN {X 0,Y 300.19,Z 419.728,A -85,B 0,C 180,E1 -16695.384,E2 -16695.384} C_VEL
LIN {X 0,Y 296.849,Z 409.793,A -85,B 0,C 180,E1 -16698.478,E2 -16698.478} C_VEL
LIN {X 0,Y 292.649,Z 398.524,A -85,B 0,C 180,E1 -16702.417,E2 -16702.417} C_VEL
LIN {X 0,Y 291.366,Z 394.81,A -85,B 0,C 180,E1 -16703.882,E2 -16703.882} C_VEL
LIN {X 0,Y 291.356,Z 394.821,A -85,B 0,C 180,E1 -16707.949,E2 -16707.949} C_VEL
LIN {X 0,Y 291.332,Z 394.824,A -85,B 0,C 180,E1 -16711.153,E2 -16711.153} C_VEL
LIN {X 0,Y 291.332,Z 394.826,A -85,B 0,C 180,E1 -16714.264,E2 -16714.264} C_VEL
LIN {X 0,Y 291.338,Z 394.824,A -85,B 0,C 180,E1 -16717.296,E2 -16717.296} C_VEL
LIN {X 0,Y 291.374,Z 394.816,A -85,B 0,C 180,E1 -16720.265,E2 -16720.265} C_VEL
LIN {X 0,Y 291.441,Z 394.809,A -85,B 0,C 180,E1 -16724.699,E2 -16724.699} C_VEL
LIN {X 0,Y 291.514,Z 394.794,A -85,B 0,C 180,E1 -16728.88,E2 -16728.88} C_VEL
LIN {X 0,Y 291.639,Z 394.783,A -85,B 0,C 180,E1 -16731.687,E2 -16731.687} C_VEL
LIN {X 0,Y 291.586,Z 394.782,A -85,B 0,C 180,E1 -16734.468,E2 -16734.468} C_VEL
LIN {X 0,Y 291.859,Z 394.751,A -85,B 0,C 180,E1 -16738.621,E2 -16738.621} C_VEL
LIN {X 0,Y 291.869,Z 394.743,A -85,B 0,C 180,E1 -16741.38,E2 -16741.38} C_VEL
LIN {X 0,Y 291.678,Z 394.735,A -85,B 0,C 180,E1 -16746.92,E2 -16746.92} C_VEL
LIN {X 0,Y 291.553,Z 394.786,A -85,B 0,C 180,E1 -16749.715,E2 -16749.715} C_VEL
LIN {X 0,Y 291.504,Z 394.765,A -85,B 0,C 180,E1 -16753.952,E2 -16753.952} C_VEL
LIN {X 0,Y 291.431,Z 394.801,A -85,B 0,C 180,E1 -16756.822,E2 -16756.822} C_VEL
LIN {X 0,Y 291.416,Z 394.785,A -85,B 0,C 180,E1 -16759.861,E2 -16759.861} C_VEL
LIN {X 0,Y 291.325,Z 394.823,A -85,B 0,C 180,E1 -16764.212,E2 -16764.212} C_VEL
LIN {X 0,Y 291.325,Z 394.798,A -85,B 0,C 180,E1 -16767.282,E2 -16767.282} C_VEL
LIN {X 0,Y 291.31,Z 394.818,A -85,B 0,C 180,E1 -16770.44,E2 -16770.44} C_VEL
LIN {X 0,Y 291.336,Z 394.816,A -85,B 0,C 180,E1 -16773.7,E2 -16773.7} C_VEL
LIN {X 0,Y 291.386,Z 394.89,A -85,B 0,C 180,E1 -16777.084,E2 -16777.084} C_VEL
LIN {X 0,Y 292.194,Z 397.333,A -85,B 0,C 180,E1 -16777.353,E2 -16777.353} C_VEL
LIN {X 0,Y 293.915,Z 399.445,A -85,B 0,C 180,E1 -16777.806,E2 -16777.806} C_VEL
LIN {X 0,Y 294.829,Z 400.391,A -85,B 0,C 180,E1 -16778.036,E2 -16778.036} C_VEL
LIN {X 0,Y 296.888,Z 403.604,A -85,B 0,C 180,E1 -16778.584,E2 -16778.584} C_VEL
LIN {X 0,Y 298.287,Z 405.38,A -85,B 0,C 180,E1 -16778.935,E2 -16778.935} C_VEL
LIN {X 0,Y 306.744,Z 417.51,A -85,B 0,C 180,E1 -16780.984,E2 -16780.984} C_VEL
LIN {X 0,Y 316.273,Z 432.439,A -85,B 0,C 180,E1 -16783.121,E2 -16783.121} C_VEL
LIN {X 0,Y 325.442,Z 448.609,A -85,B 0,C 180,E1 -16785.042,E2 -16785.042} C_VEL
LIN {X 0,Y 322.869,Z 514.36,A -85,B 0,C 180,E1 -16786.526,E2 -16786.526} C_VEL
LIN {X 0,Y 322.317,Z 533.02,A -85,B 0,C 180,E1 -16787.06,E2 -16787.06} C_VEL
LIN {X 0,Y 321.385,Z 547.65,A -85,B 0,C 180,E1 -16787.707,E2 -16787.707} C_VEL
LIN {X 0,Y 320.051,Z 560.616,A -85,B 0,C 180,E1 -16788.47,E2 -16788.47} C_VEL
LIN {X 0,Y 318.229,Z 574.639,A -85,B 0,C 180,E1 -16789.555,E2 -16789.555} C_VEL
LIN {X 0,Y 315.912,Z 588.296,A -85,B 0,C 180,E1 -16790.881,E2 -16790.881} C_VEL
LIN {X 0,Y 313.386,Z 600.705,A -85,B 0,C 180,E1 -16792.366,E2 -16792.366} C_VEL
LIN {X 0,Y 310.794,Z 611.854,A -85,B 0,C 180,E1 -16793.991,E2 -16793.991} C_VEL
LIN {X 0,Y 307.834,Z 623.231,A -85,B 0,C 180,E1 -16795.991,E2 -16795.991} C_VEL
LIN {X 0,Y 304.78,Z 633.809,A -85,B 0,C 180,E1 -16798.263,E2 -16798.263} C_VEL
LIN {X 0,Y 301.852,Z 643.126,A -85,B 0,C 180,E1 -16800.73,E2 -16800.73} C_VEL
LIN {X 0,Y 299.492,Z 650.323,A -85,B 0,C 180,E1 -16803.092,E2 -16803.092} C_VEL
LIN {X 0,Y 297.359,Z 656.466,A -85,B 0,C 180,E1 -16805.57,E2 -16805.57} C_VEL
LIN {X 0,Y 295.666,Z 661.235,A -85,B 0,C 180,E1 -16807.978,E2 -16807.978} C_VEL
LIN {X 0,Y 294.272,Z 665.082,A -85,B 0,C 180,E1 -16810.468,E2 -16810.468} C_VEL
LIN {X 0,Y 293.073,Z 668.156,A -85,B 0,C 180,E1 -16813.277,E2 -16813.277} C_VEL
LIN {X 0,Y 292.248,Z 670.027,A -85,B 0,C 180,E1 -16816.086,E2 -16816.086} C_VEL
LIN {X 0,Y 291.863,Z 670.752,A -85,B 0,C 180,E1 -16818.894,E2 -16818.894} C_VEL
LIN {X 0,Y 291.763,Z 670.376,A -85,B 0,C 180,E1 -16821.691,E2 -16821.691} C_VEL
LIN {X 0,Y 291.742,Z 668.94,A -85,B 0,C 180,E1 -16824.471,E2 -16824.471} C_VEL
LIN {X 0,Y 292.159,Z 666.353,A -85,B 0,C 180,E1 -16827.243,E2 -16827.243} C_VEL
LIN {X 0,Y 292.897,Z 662.55,A -85,B 0,C 180,E1 -16830.001,E2 -16830.001} C_VEL
LIN {X 0,Y 293.898,Z 657.511,A -85,B 0,C 180,E1 -16832.742,E2 -16832.742} C_VEL
LIN {X 0,Y 295.298,Z 651.086,A -85,B 0,C 180,E1 -16835.463,E2 -16835.463} C_VEL
LIN {X 0,Y 296.748,Z 644.187,A -85,B 0,C 180,E1 -16837.827,E2 -16837.827} C_VEL
LIN {X 0,Y 298.57,Z 635.889,A -85,B 0,C 180,E1 -16840.169,E2 -16840.169} C_VEL
LIN {X 0,Y 300.703,Z 625.913,A -85,B 0,C 180,E1 -16842.486,E2 -16842.486} C_VEL
LIN {X 0,Y 302.701,Z 615.729,A -85,B 0,C 180,E1 -16844.453,E2 -16844.453} C_VEL
LIN {X 0,Y 304.606,Z 604.694,A -85,B 0,C 180,E1 -16846.246,E2 -16846.246} C_VEL
LIN {X 0,Y 306.58,Z 592.694,A -85,B 0,C 180,E1 -16847.855,E2 -16847.855} C_VEL
LIN {X 0,Y 308.453,Z 579.587,A -85,B 0,C 180,E1 -16849.292,E2 -16849.292} C_VEL
LIN {X 0,Y 310.243,Z 564.997,A -85,B 0,C 180,E1 -16850.556,E2 -16850.556} C_VEL
LIN {X 0,Y 311.619,Z 549.601,A -85,B 0,C 180,E1 -16851.578,E2 -16851.578} C_VEL
LIN {X 0,Y 312.498,Z 534.972,A -85,B 0,C 180,E1 -16852.29,E2 -16852.29} C_VEL
LIN {X 0,Y 312.909,Z 519.961,A -85,B 0,C 180,E1 -16852.779,E2 -16852.779} C_VEL
LIN {X 0,Y 315.077,Z 447.389,A -85,B 0,C 180,E1 -16854.439,E2 -16854.439} C_VEL
LIN {X 0,Y 315.224,Z 440.263,A -85,B 0,C 180,E1 -16854.609,E2 -16854.609} C_VEL
LIN {X 0,Y 308.197,Z 425.678,A -85,B 0,C 180,E1 -16855.798,E2 -16855.798} C_VEL
LIN {X 0,Y 299.222,Z 409.038,A -85,B 0,C 180,E1 -16857.363,E2 -16857.363} C_VEL
LIN {X 0,Y 292.935,Z 398.506,A -85,B 0,C 180,E1 -16858.5,E2 -16858.5} C_VEL
LIN {X 0,Y 291.495,Z 395.724,A -85,B 0,C 180,E1 -16858.78,E2 -16858.78} C_VEL
LIN {X 0,Y 291.314,Z 394.811,A -85,B 0,C 180,E1 -16858.849,E2 -16858.849} C_VEL
LIN {X 0,Y 291.339,Z 394.822,A -85,B 0,C 180,E1 -16862.401,E2 -16862.401} C_VEL
LIN {X 0,Y 291.355,Z 394.819,A -85,B 0,C 180,E1 -16865.374,E2 -16865.374} C_VEL
LIN {X 0,Y 291.309,Z 394.824,A -85,B 0,C 180,E1 -16868.848,E2 -16868.848} C_VEL
LIN {X 0,Y 291.282,Z 394.827,A -85,B 0,C 180,E1 -16872.498,E2 -16872.498} C_VEL
LIN {X 0,Y 291.286,Z 394.825,A -85,B 0,C 180,E1 -16876.37,E2 -16876.37} C_VEL
LIN {X 0,Y 291.286,Z 394.821,A -85,B 0,C 180,E1 -16878.272,E2 -16878.272} C_VEL
LIN {X 0,Y 290.652,Z 394.909,A -85,B 0,C 180,E1 -16879.427,E2 -16879.427} C_VEL
LIN {X 0,Y 287.809,Z 395.263,A -85,B 0,C 180,E1 -16881.309,E2 -16881.309} C_VEL
LIN {X 0,Y 285.396,Z 395.561,A -85,B 0,C 180,E1 -16882.836,E2 -16882.836} C_VEL
LIN {X 0,Y 284.388,Z 395.688,A -85,B 0,C 180,E1 -16884.02,E2 -16884.02} C_VEL
LIN {X 0,Y 284.322,Z 395.695,A -85,B 0,C 180,E1 -16884.42,E2 -16884.42} C_VEL
LIN {X 0,Y 284.273,Z 395.702,A -85,B 0,C 180,E1 -16888.722,E2 -16888.722} C_VEL
LIN {X 0,Y 284.257,Z 395.698,A -85,B 0,C 180,E1 -16891.981,E2 -16891.981} C_VEL
LIN {X 0,Y 284.317,Z 395.683,A -85,B 0,C 180,E1 -16896.147,E2 -16896.147} C_VEL
LIN {X 0,Y 284.33,Z 395.687,A -85,B 0,C 180,E1 -16899.927,E2 -16899.927} C_VEL
LIN {X 0,Y 284.442,Z 395.677,A -85,B 0,C 180,E1 -16904.493,E2 -16904.493} C_VEL
LIN {X 0,Y 284.46,Z 395.624,A -85,B 0,C 180,E1 -16908.6,E2 -16908.6} C_VEL
LIN {X 0,Y 284.575,Z 395.632,A -85,B 0,C 180,E1 -16911.478,E2 -16911.478} C_VEL
LIN {X 0,Y 284.557,Z 395.663,A -85,B 0,C 180,E1 -16914.33,E2 -16914.33} C_VEL
LIN {X 0,Y 284.832,Z 395.616,A -85,B 0,C 180,E1 -16918.586,E2 -16918.586} C_VEL
LIN {X 0,Y 284.831,Z 395.63,A -85,B 0,C 180,E1 -16921.414,E2 -16921.414} C_VEL
LIN {X 0,Y 284.632,Z 395.654,A -85,B 0,C 180,E1 -16927.091,E2 -16927.091} C_VEL
LIN {X 0,Y 284.508,Z 395.66,A -85,B 0,C 180,E1 -16929.957,E2 -16929.957} C_VEL
LIN {X 0,Y 284.403,Z 395.672,A -85,B 0,C 180,E1 -16934.306,E2 -16934.306} C_VEL
LIN {X 0,Y 284.332,Z 395.694,A -85,B 0,C 180,E1 -16937.254,E2 -16937.254} C_VEL
LIN {X 0,Y 284.317,Z 395.695,A -85,B 0,C 180,E1 -16940.246,E2 -16940.246} C_VEL
LIN {X 0,Y 284.292,Z 395.694,A -85,B 0,C 180,E1 -16943.842,E2 -16943.842} C_VEL
LIN {X 0,Y 284.28,Z 395.695,A -85,B 0,C 180,E1 -16947.129,E2 -16947.129} C_VEL
LIN {X 0,Y 284.269,Z 395.698,A -85,B 0,C 180,E1 -16950.084,E2 -16950.084} C_VEL
LIN {X 0,Y 284.3,Z 395.682,A -85,B 0,C 180,E1 -16952.946,E2 -16952.946} C_VEL
LIN {X 0,Y 284.312,Z 395.699,A -85,B 0,C 180,E1 -16956.389,E2 -16956.389} C_VEL
LIN {X 0,Y 284.278,Z 395.695,A -85,B 0,C 180,E1 -16959.999,E2 -16959.999} C_VEL
LIN {X 0,Y 284.269,Z 395.79,A -85,B 0,C 180,E1 -16961.876,E2 -16961.876} C_VEL
LIN {X 0,Y 288.879,Z 410.235,A -85,B 0,C 180,E1 -16965.864,E2 -16965.864} C_VEL
LIN {X 0,Y 292.501,Z 423.479,A -85,B 0,C 180,E1 -16969.183,E2 -16969.183} C_VEL
LIN {X 0,Y 295.224,Z 434.54,A -85,B 0,C 180,E1 -16971.775,E2 -16971.775} C_VEL
LIN {X 0,Y 299.411,Z 444.938,A -85,B 0,C 180,E1 -16972.599,E2 -16972.599} C_VEL
LIN {X 0,Y 302.842,Z 472.24,A -85,B 0,C 180,E1 -16973.767,E2 -16973.767} C_VEL
LIN {X 0,Y 307.524,Z 514.377,A -85,B 0,C 180,E1 -16975.429,E2 -16975.429} C_VEL
LIN {X 0,Y 304.37,Z 605.062,A -85,B 0,C 180,E1 -16977.531,E2 -16977.531} C_VEL
LIN {X 0,Y 303.164,Z 620.592,A -85,B 0,C 180,E1 -16978.122,E2 -16978.122} C_VEL
LIN {X 0,Y 301.417,Z 635.623,A -85,B 0,C 180,E1 -16978.944,E2 -16978.944} C_VEL
LIN {X 0,Y 299.077,Z 650.693,A -85,B 0,C 180,E1 -16980.043,E2 -16980.043} C_VEL
LIN {X 0,Y 296.652,Z 663.956,A -85,B 0,C 180,E1 -16981.288,E2 -16981.288} C_VEL
LIN {X 0,Y 294.282,Z 676.972,A -85,B 0,C 180,E1 -16982.823,E2 -16982.823} C_VEL
LIN {X 0,Y 291.875,Z 688.746,A -85,B 0,C 180,E1 -16984.507,E2 -16984.507} C_VEL
LIN {X 0,Y 289.62,Z 699.746,A -85,B 0,C 180,E1 -16986.397,E2 -16986.397} C_VEL
LIN {X 0,Y 287.564,Z 709.953,A -85,B 0,C 180,E1 -16988.494,E2 -16988.494} C_VEL
LIN {X 0,Y 285.8,Z 720.001,A -85,B 0,C 180,E1 -16990.984,E2 -16990.984} C_VEL
LIN {X 0,Y 284.447,Z 728.383,A -85,B 0,C 180,E1 -16993.493,E2 -16993.493} C_VEL
LIN {X 0,Y 283.612,Z 736.251,A -85,B 0,C 180,E1 -16996.384,E2 -16996.384} C_VEL
LIN {X 0,Y 283.306,Z 742.518,A -85,B 0,C 180,E1 -16999.277,E2 -16999.277} C_VEL
LIN {X 0,Y 283.433,Z 746.258,A -85,B 0,C 180,E1 -17001.444,E2 -17001.444} C_VEL
LIN {X 0,Y 283.781,Z 750.041,A -85,B 0,C 180,E1 -17004.314,E2 -17004.314} C_VEL
LIN {X 0,Y 284.035,Z 752.479,A -85,B 0,C 180,E1 -17007.163,E2 -17007.163} C_VEL
LIN {X 0,Y 284.354,Z 753.249,A -85,B 0,C 180,E1 -17008.583,E2 -17008.583} C_VEL
LIN {X 0,Y 284.599,Z 753.699,A -85,B 0,C 180,E1 -17009.999,E2 -17009.999} C_VEL
LIN {X 0,Y 284.318,Z 753.758,A -85,B 0,C 180,E1 -17011.416,E2 -17011.416} C_VEL
LIN {X 0,Y 283.833,Z 752.919,A -85,B 0,C 180,E1 -17014.259,E2 -17014.259} C_VEL
LIN {X 0,Y 283.37,Z 750.772,A -85,B 0,C 180,E1 -17017.228,E2 -17017.228} C_VEL
LIN {X 0,Y 283.101,Z 746.605,A -85,B 0,C 180,E1 -17020.73,E2 -17020.73} C_VEL
LIN {X 0,Y 283.448,Z 741.757,A -85,B 0,C 180,E1 -17023.623,E2 -17023.623} C_VEL
LIN {X 0,Y 284.438,Z 735.566,A -85,B 0,C 180,E1 -17026.507,E2 -17026.507} C_VEL
LIN {X 0,Y 286.164,Z 727.898,A -85,B 0,C 180,E1 -17029.362,E2 -17029.362} C_VEL
LIN {X 0,Y 288.395,Z 718.992,A -85,B 0,C 180,E1 -17032.055,E2 -17032.055} C_VEL
LIN {X 0,Y 291.303,Z 708.679,A -85,B 0,C 180,E1 -17034.592,E2 -17034.592} C_VEL
LIN {X 0,Y 294.099,Z 698.719,A -85,B 0,C 180,E1 -17036.618,E2 -17036.618} C_VEL
LIN {X 0,Y 297.533,Z 687.006,A -85,B 0,C 180,E1 -17038.575,E2 -17038.575} C_VEL
LIN {X 0,Y 300.986,Z 674.058,A -85,B 0,C 180,E1 -17040.344,E2 -17040.344} C_VEL
LIN {X 0,Y 304.101,Z 661.615,A -85,B 0,C 180,E1 -17041.719,E2 -17041.719} C_VEL
LIN {X 0,Y 307.218,Z 648.066,A -85,B 0,C 180,E1 -17042.908,E2 -17042.908} C_VEL
LIN {X 0,Y 310.113,Z 633.093,A -85,B 0,C 180,E1 -17043.921,E2 -17043.921} C_VEL
LIN {X 0,Y 312.29,Z 618.237,A -85,B 0,C 180,E1 -17044.675,E2 -17044.675} C_VEL
LIN {X 0,Y 313.766,Z 603.011,A -85,B 0,C 180,E1 -17045.222,E2 -17045.222} C_VEL
LIN {X 0,Y 317.501,Z 516.398,A -85,B 0,C 180,E1 -17047.206,E2 -17047.206} C_VEL
LIN {X 0,Y 315.564,Z 496.508,A -85,B 0,C 180,E1 -17048.083,E2 -17048.083} C_VEL
LIN {X 0,Y 312.011,Z 469.519,A -85,B 0,C 180,E1 -17049.463,E2 -17049.463} C_VEL
LIN {X 0,Y 310.109,Z 457.483,A -85,B 0,C 180,E1 -17050.153,E2 -17050.153} C_VEL
LIN {X 0,Y 302.08,Z 440.984,A -85,B 0,C 180,E1 -17052.121,E2 -17052.121} C_VEL
LIN {X 0,Y 297.933,Z 433.35,A -85,B 0,C 180,E1 -17053.179,E2 -17053.179} C_VEL
LIN {X 0,Y 295.959,Z 429.378,A -85,B 0,C 180,E1 -17053.743,E2 -17053.743} C_VEL
LIN {X 0,Y 292.53,Z 418.342,A -85,B 0,C 180,E1 -17057.074,E2 -17057.074} C_VEL
LIN {X 0,Y 289.096,Z 408.594,A -85,B 0,C 180,E1 -17060.347,E2 -17060.347} C_VEL
LIN {X 0,Y 285.657,Z 399.294,A -85,B 0,C 180,E1 -17063.81,E2 -17063.81} C_VEL
LIN {X 0,Y 284.3,Z 395.698,A -85,B 0,C 180,E1 -17065.35,E2 -17065.35} C_VEL
LIN {X 0,Y 284.275,Z 395.697,A -85,B 0,C 180,E1 -17068.724,E2 -17068.724} C_VEL
LIN {X 0,Y 284.264,Z 395.698,A -85,B 0,C 180,E1 -17071.983,E2 -17071.983} C_VEL
LIN {X 0,Y 284.282,Z 395.695,A -85,B 0,C 180,E1 -17076.16,E2 -17076.16} C_VEL
LIN {X 0,Y 284.324,Z 395.691,A -85,B 0,C 180,E1 -17079.928,E2 -17079.928} C_VEL
LIN {X 0,Y 284.41,Z 395.686,A -85,B 0,C 180,E1 -17084.512,E2 -17084.512} C_VEL
LIN {X 0,Y 284.446,Z 395.677,A -85,B 0,C 180,E1 -17088.6,E2 -17088.6} C_VEL
LIN {X 0,Y 284.597,Z 395.66,A -85,B 0,C 180,E1 -17091.48,E2 -17091.48} C_VEL
LIN {X 0,Y 284.556,Z 395.657,A -85,B 0,C 180,E1 -17094.331,E2 -17094.331} C_VEL
LIN {X 0,Y 284.826,Z 395.626,A -85,B 0,C 180,E1 -17098.586,E2 -17098.586} C_VEL
LIN {X 0,Y 284.835,Z 395.62,A -85,B 0,C 180,E1 -17101.414,E2 -17101.414} C_VEL
LIN {X 0,Y 284.63,Z 395.612,A -85,B 0,C 180,E1 -17107.092,E2 -17107.092} C_VEL
LIN {X 0,Y 284.501,Z 395.668,A -85,B 0,C 180,E1 -17109.958,E2 -17109.958} C_VEL
LIN {X 0,Y 284.453,Z 395.641,A -85,B 0,C 180,E1 -17114.305,E2 -17114.305} C_VEL
LIN {X 0,Y 284.365,Z 395.679,A -85,B 0,C 180,E1 -17118.741,E2 -17118.741} C_VEL
LIN {X 0,Y 284.293,Z 395.67,A -85,B 0,C 180,E1 -17121.766,E2 -17121.766} C_VEL
LIN {X 0,Y 284.28,Z 395.693,A -85,B 0,C 180,E1 -17124.852,E2 -17124.852} C_VEL
LIN {X 0,Y 284.265,Z 395.684,A -85,B 0,C 180,E1 -17128.018,E2 -17128.018} C_VEL
LIN {X 0,Y 284.277,Z 395.683,A -85,B 0,C 180,E1 -17131.277,E2 -17131.277} C_VEL
LIN {X 0,Y 284.337,Z 395.87,A -85,B 0,C 180,E1 -17135.478,E2 -17135.478} C_VEL
LIN {X 0,Y 285.282,Z 398.485,A -85,B 0,C 180,E1 -17135.807,E2 -17135.807} C_VEL
LIN {X 0,Y 287.351,Z 400.656,A -85,B 0,C 180,E1 -17136.378,E2 -17136.378} C_VEL
LIN {X 0,Y 288.23,Z 401.928,A -85,B 0,C 180,E1 -17136.629,E2 -17136.629} C_VEL
LIN {X 0,Y 290.394,Z 404.967,A -85,B 0,C 180,E1 -17137.232,E2 -17137.232} C_VEL
LIN {X 0,Y 291.739,Z 406.799,A -85,B 0,C 180,E1 -17137.597,E2 -17137.597} C_VEL
LIN {X 0,Y 295.569,Z 412.221,A -85,B 0,C 180,E1 -17138.611,E2 -17138.611} C_VEL
LIN {X 0,Y 301.204,Z 420.268,A -85,B 0,C 180,E1 -17140.025,E2 -17140.025} C_VEL
LIN {X 0,Y 309.7,Z 433.371,A -85,B 0,C 180,E1 -17142.024,E2 -17142.024} C_VEL
LIN {X 0,Y 318.049,Z 447.766,A -85,B 0,C 180,E1 -17143.87,E2 -17143.87} C_VEL
LIN {X 0,Y 319.975,Z 451.376,A -85,B 0,C 180,E1 -17144.282,E2 -17144.282} C_VEL
LIN {X 0,Y 317.371,Z 514.231,A -85,B 0,C 180,E1 -17145.713,E2 -17145.713} C_VEL
LIN {X 0,Y 316.788,Z 533.604,A -85,B 0,C 180,E1 -17146.27,E2 -17146.27} C_VEL
LIN {X 0,Y 315.802,Z 548.286,A -85,B 0,C 180,E1 -17146.919,E2 -17146.919} C_VEL
LIN {X 0,Y 314.421,Z 561.474,A -85,B 0,C 180,E1 -17147.704,E2 -17147.704} C_VEL
LIN {X 0,Y 312.429,Z 576.096,A -85,B 0,C 180,E1 -17148.857,E2 -17148.857} C_VEL
LIN {X 0,Y 310.061,Z 589.519,A -85,B 0,C 180,E1 -17150.186,E2 -17150.186} C_VEL
LIN {X 0,Y 307.174,Z 603.017,A -85,B 0,C 180,E1 -17151.85,E2 -17151.85} C_VEL
LIN {X 0,Y 304.491,Z 614.027,A -85,B 0,C 180,E1 -17153.505,E2 -17153.505} C_VEL
LIN {X 0,Y 301.368,Z 625.33,A -85,B 0,C 180,E1 -17155.563,E2 -17155.563} C_VEL
LIN {X 0,Y 298.234,Z 635.617,A -85,B 0,C 180,E1 -17157.856,E2 -17157.856} C_VEL
LIN {X 0,Y 295.174,Z 644.842,A -85,B 0,C 180,E1 -17160.394,E2 -17160.394} C_VEL
LIN {X 0,Y 292.667,Z 652.092,A -85,B 0,C 180,E1 -17162.855,E2 -17162.855} C_VEL
LIN {X 0,Y 290.25,Z 658.741,A -85,B 0,C 180,E1 -17165.694,E2 -17165.694} C_VEL
LIN {X 0,Y 288.287,Z 663.878,A -85,B 0,C 180,E1 -17168.552,E2 -17168.552} C_VEL
LIN {X 0,Y 286.799,Z 667.638,A -85,B 0,C 180,E1 -17171.425,E2 -17171.425} C_VEL
LIN {X 0,Y 285.734,Z 670.154,A -85,B 0,C 180,E1 -17174.303,E2 -17174.303} C_VEL
LIN {X 0,Y 285.059,Z 671.508,A -85,B 0,C 180,E1 -17177.181,E2 -17177.181} C_VEL
LIN {X 0,Y 284.782,Z 671.737,A -85,B 0,C 180,E1 -17180.053,E2 -17180.053} C_VEL
LIN {X 0,Y 284.795,Z 670.874,A -85,B 0,C 180,E1 -17182.913,E2 -17182.913} C_VEL
LIN {X 0,Y 284.913,Z 668.931,A -85,B 0,C 180,E1 -17185.757,E2 -17185.757} C_VEL
LIN {X 0,Y 285.444,Z 665.788,A -85,B 0,C 180,E1 -17188.59,E2 -17188.59} C_VEL
LIN {X 0,Y 286.271,Z 661.453,A -85,B 0,C 180,E1 -17191.407,E2 -17191.407} C_VEL
LIN {X 0,Y 287.529,Z 655.804,A -85,B 0,C 180,E1 -17194.206,E2 -17194.206} C_VEL
LIN {X 0,Y 289.175,Z 648.692,A -85,B 0,C 180,E1 -17196.98,E2 -17196.98} C_VEL
LIN {X 0,Y 290.845,Z 641.104,A -85,B 0,C 180,E1 -17199.388,E2 -17199.388} C_VEL
LIN {X 0,Y 292.934,Z 631.976,A -85,B 0,C 180,E1 -17201.767,E2 -17201.767} C_VEL
LIN {X 0,Y 294.928,Z 622.711,A -85,B 0,C 180,E1 -17203.786,E2 -17203.786} C_VEL
LIN {X 0,Y 297.086,Z 611.729,A -85,B 0,C 180,E1 -17205.786,E2 -17205.786} C_VEL
LIN {X 0,Y 299.104,Z 599.715,A -85,B 0,C 180,E1 -17207.609,E2 -17207.609} C_VEL
LIN {X 0,Y 301.343,Z 586.368,A -85,B 0,C 180,E1 -17209.234,E2 -17209.234} C_VEL
LIN {X 0,Y 303.05,Z 573.346,A -85,B 0,C 180,E1 -17210.534,E2 -17210.534} C_VEL
LIN {X 0,Y 304.681,Z 558.904,A -85,B 0,C 180,E1 -17211.658,E2 -17211.658} C_VEL
LIN {X 0,Y 305.865,Z 543.874,A -85,B 0,C 180,E1 -17212.546,E2 -17212.546} C_VEL
LIN {X 0,Y 306.549,Z 528.071,A -85,B 0,C 180,E1 -17213.201,E2 -17213.201} C_VEL
LIN {X 0,Y 307.598,Z 487.762,A -85,B 0,C 180,E1 -17214.195,E2 -17214.195} C_VEL
LIN {X 0,Y 309.106,Z 442.306,A -85,B 0,C 180,E1 -17215.244,E2 -17215.244} C_VEL
LIN {X 0,Y 301.545,Z 426.835,A -85,B 0,C 180,E1 -17216.569,E2 -17216.569} C_VEL
LIN {X 0,Y 292.478,Z 410.243,A -85,B 0,C 180,E1 -17218.217,E2 -17218.217} C_VEL
LIN {X 0,Y 285.92,Z 399.412,A -85,B 0,C 180,E1 -17219.459,E2 -17219.459} C_VEL
LIN {X 0,Y 284.482,Z 396.654,A -85,B 0,C 180,E1 -17219.754,E2 -17219.754} C_VEL
LIN {X 0,Y 284.292,Z 395.678,A -85,B 0,C 180,E1 -17219.873,E2 -17219.873} C_VEL
LIN {X 0,Y 284.305,Z 395.696,A -85,B 0,C 180,E1 -17222.945,E2 -17222.945} C_VEL
LIN {X 0,Y 284.32,Z 395.69,A -85,B 0,C 180,E1 -17226.387,E2 -17226.387} C_VEL
LIN {X 0,Y 284.254,Z 395.694,A -85,B 0,C 180,E1 -17230.003,E2 -17230.003} C_VEL
LIN {X 0,Y 284.231,Z 395.699,A -85,B 0,C 180,E1 -17234.187,E2 -17234.187} C_VEL
LIN {X 0,Y 284.227,Z 395.699,A -85,B 0,C 180,E1 -17238.255,E2 -17238.255} C_VEL
LIN {X 0,Y 284.28,Z 395.693,A -85,B 0,C 180,E1 -17242.288,E2 -17242.288} C_VEL
LIN {X 0,Y 284.322,Z 395.695,A -85,B 0,C 180,E1 -17244.42,E2 -17244.42} C_VEL
LIN {X 0,Y 283.68,Z 395.776,A -85,B 0,C 180,E1 -17245.602,E2 -17245.602} C_VEL
LIN {X 0,Y 280.784,Z 396.133,A -85,B 0,C 180,E1 -17247.524,E2 -17247.524} C_VEL
LIN {X 0,Y 278.314,Z 396.445,A -85,B 0,C 180,E1 -17249.086,E2 -17249.086} C_VEL
LIN {X 0,Y 277.268,Z 396.566,A -85,B 0,C 180,E1 -17250.298,E2 -17250.298} C_VEL
LIN {X 0,Y 277.192,Z 396.572,A -85,B 0,C 180,E1 -17250.708,E2 -17250.708} C_VEL
LIN {X 0,Y 277.241,Z 396.575,A -85,B 0,C 180,E1 -17254.472,E2 -17254.472} C_VEL
LIN {X 0,Y 277.255,Z 396.573,A -85,B 0,C 180,E1 -17257.652,E2 -17257.652} C_VEL
LIN {X 0,Y 277.28,Z 396.56,A -85,B 0,C 180,E1 -17260.761,E2 -17260.761} C_VEL
LIN {X 0,Y 277.404,Z 396.547,A -85,B 0,C 180,E1 -17265.324,E2 -17265.324} C_VEL
LIN {X 0,Y 277.448,Z 396.496,A -85,B 0,C 180,E1 -17269.786,E2 -17269.786} C_VEL
LIN {X 0,Y 277.585,Z 396.522,A -85,B 0,C 180,E1 -17272.727,E2 -17272.727} C_VEL
LIN {X 0,Y 277.797,Z 396.492,A -85,B 0,C 180,E1 -17278.55,E2 -17278.55} C_VEL
LIN {X 0,Y 277.798,Z 396.505,A -85,B 0,C 180,E1 -17281.449,E2 -17281.449} C_VEL
LIN {X 0,Y 277.591,Z 396.531,A -85,B 0,C 180,E1 -17287.272,E2 -17287.272} C_VEL
LIN {X 0,Y 277.448,Z 396.541,A -85,B 0,C 180,E1 -17290.213,E2 -17290.213} C_VEL
LIN {X 0,Y 277.361,Z 396.55,A -85,B 0,C 180,E1 -17294.678,E2 -17294.678} C_VEL
LIN {X 0,Y 277.267,Z 396.564,A -85,B 0,C 180,E1 -17299.239,E2 -17299.239} C_VEL
LIN {X 0,Y 277.254,Z 396.571,A -85,B 0,C 180,E1 -17303.927,E2 -17303.927} C_VEL
LIN {X 0,Y 277.23,Z 396.575,A -85,B 0,C 180,E1 -17307.469,E2 -17307.469} C_VEL
LIN {X 0,Y 277.224,Z 396.579,A -85,B 0,C 180,E1 -17310.466,E2 -17310.466} C_VEL
LIN {X 0,Y 277.241,Z 396.557,A -85,B 0,C 180,E1 -17313.896,E2 -17313.896} C_VEL
LIN {X 0,Y 277.244,Z 396.567,A -85,B 0,C 180,E1 -17317.473,E2 -17317.473} C_VEL
LIN {X 0,Y 277.245,Z 396.784,A -85,B 0,C 180,E1 -17321.012,E2 -17321.012} C_VEL
LIN {X 0,Y 281.08,Z 408.597,A -85,B 0,C 180,E1 -17324.435,E2 -17324.435} C_VEL
LIN {X 0,Y 284.276,Z 419.509,A -85,B 0,C 180,E1 -17327.349,E2 -17327.349} C_VEL
LIN {X 0,Y 287.776,Z 433.304,A -85,B 0,C 180,E1 -17330.747,E2 -17330.747} C_VEL
LIN {X 0,Y 293.649,Z 447.494,A -85,B 0,C 180,E1 -17331.944,E2 -17331.944} C_VEL
LIN {X 0,Y 296.93,Z 474.466,A -85,B 0,C 180,E1 -17333.123,E2 -17333.123} C_VEL
LIN {X 0,Y 301.373,Z 515.272,A -85,B 0,C 180,E1 -17334.774,E2 -17334.774} C_VEL
LIN {X 0,Y 298.147,Z 604.075,A -85,B 0,C 180,E1 -17336.868,E2 -17336.868} C_VEL
LIN {X 0,Y 296.874,Z 619.581,A -85,B 0,C 180,E1 -17337.464,E2 -17337.464} C_VEL
LIN {X 0,Y 295.124,Z 634.627,A -85,B 0,C 180,E1 -17338.306,E2 -17338.306} C_VEL
LIN {X 0,Y 292.956,Z 648.724,A -85,B 0,C 180,E1 -17339.351,E2 -17339.351} C_VEL
LIN {X 0,Y 290.325,Z 662.514,A -85,B 0,C 180,E1 -17340.647,E2 -17340.647} C_VEL
LIN {X 0,Y 287.834,Z 675.286,A -85,B 0,C 180,E1 -17342.162,E2 -17342.162} C_VEL
LIN {X 0,Y 285.409,Z 687.194,A -85,B 0,C 180,E1 -17343.886,E2 -17343.886} C_VEL
LIN {X 0,Y 282.998,Z 698.272,A -85,B 0,C 180,E1 -17345.81,E2 -17345.81} C_VEL
LIN {X 0,Y 280.862,Z 708.56,A -85,B 0,C 180,E1 -17347.954,E2 -17347.954} C_VEL
LIN {X 0,Y 278.953,Z 718.665,A -85,B 0,C 180,E1 -17350.499,E2 -17350.499} C_VEL
LIN {X 0,Y 277.522,Z 727.104,A -85,B 0,C 180,E1 -17353.068,E2 -17353.068} C_VEL
LIN {X 0,Y 276.609,Z 735.022,A -85,B 0,C 180,E1 -17356.032,E2 -17356.032} C_VEL
LIN {X 0,Y 276.245,Z 741.336,A -85,B 0,C 180,E1 -17359,E2 -17359} C_VEL
LIN {X 0,Y 276.354,Z 745.101,A -85,B 0,C 180,E1 -17361.223,E2 -17361.223} C_VEL
LIN {X 0,Y 276.722,Z 748.934,A -85,B 0,C 180,E1 -17364.169,E2 -17364.169} C_VEL
LIN {X 0,Y 276.991,Z 751.414,A -85,B 0,C 180,E1 -17367.091,E2 -17367.091} C_VEL
LIN {X 0,Y 277.321,Z 752.205,A -85,B 0,C 180,E1 -17368.547,E2 -17368.547} C_VEL
LIN {X 0,Y 277.577,Z 752.674,A -85,B 0,C 180,E1 -17369.999,E2 -17369.999} C_VEL
LIN {X 0,Y 277.282,Z 752.736,A -85,B 0,C 180,E1 -17371.452,E2 -17371.452} C_VEL
LIN {X 0,Y 276.783,Z 751.923,A -85,B 0,C 180,E1 -17374.368,E2 -17374.368} C_VEL
LIN {X 0,Y 276.291,Z 749.897,A -85,B 0,C 180,E1 -17377.306,E2 -17377.306} C_VEL
LIN {X 0,Y 276.033,Z 746.665,A -85,B 0,C 180,E1 -17380.266,E2 -17380.266} C_VEL
LIN {X 0,Y 276.282,Z 742.202,A -85,B 0,C 180,E1 -17383.234,E2 -17383.234} C_VEL
LIN {X 0,Y 277.2,Z 736.423,A -85,B 0,C 180,E1 -17386.193,E2 -17386.193} C_VEL
LIN {X 0,Y 278.81,Z 729.186,A -85,B 0,C 180,E1 -17389.128,E2 -17389.128} C_VEL
LIN {X 0,Y 281.181,Z 720.33,A -85,B 0,C 180,E1 -17392.018,E2 -17392.018} C_VEL
LIN {X 0,Y 283.892,Z 711.008,A -85,B 0,C 180,E1 -17394.497,E2 -17394.497} C_VEL
LIN {X 0,Y 287.18,Z 699.907,A -85,B 0,C 180,E1 -17396.918,E2 -17396.918} C_VEL
LIN {X 0,Y 290.959,Z 687.565,A -85,B 0,C 180,E1 -17399.084,E2 -17399.084} C_VEL
LIN {X 0,Y 294.734,Z 674.062,A -85,B 0,C 180,E1 -17400.994,E2 -17400.994} C_VEL
LIN {X 0,Y 298.07,Z 661.353,A -85,B 0,C 180,E1 -17402.438,E2 -17402.438} C_VEL
LIN {X 0,Y 301.289,Z 647.956,A -85,B 0,C 180,E1 -17403.64,E2 -17403.64} C_VEL
LIN {X 0,Y 304.261,Z 633.274,A -85,B 0,C 180,E1 -17404.665,E2 -17404.665} C_VEL
LIN {X 0,Y 306.587,Z 618.03,A -85,B 0,C 180,E1 -17405.466,E2 -17405.466} C_VEL
LIN {X 0,Y 308.134,Z 603.168,A -85,B 0,C 180,E1 -17406.015,E2 -17406.015} C_VEL
LIN {X 0,Y 310.198,Z 558.672,A -85,B 0,C 180,E1 -17407.076,E2 -17407.076} C_VEL
LIN {X 0,Y 312.01,Z 516.842,A -85,B 0,C 180,E1 -17408.037,E2 -17408.037} C_VEL
LIN {X 0,Y 310.154,Z 497.438,A -85,B 0,C 180,E1 -17408.919,E2 -17408.919} C_VEL
LIN {X 0,Y 306.747,Z 470.926,A -85,B 0,C 180,E1 -17410.313,E2 -17410.313} C_VEL
LIN {X 0,Y 305.154,Z 460.832,A -85,B 0,C 180,E1 -17410.914,E2 -17410.914} C_VEL
LIN {X 0,Y 297.882,Z 445.614,A -85,B 0,C 180,E1 -17412.772,E2 -17412.772} C_VEL
LIN {X 0,Y 291.392,Z 433.441,A -85,B 0,C 180,E1 -17414.519,E2 -17414.519} C_VEL
LIN {X 0,Y 288.328,Z 427.753,A -85,B 0,C 180,E1 -17415.413,E2 -17415.413} C_VEL
LIN {X 0,Y 284.995,Z 417.503,A -85,B 0,C 180,E1 -17418.727,E2 -17418.727} C_VEL
LIN {X 0,Y 281.436,Z 407.68,A -85,B 0,C 180,E1 -17422.28,E2 -17422.28} C_VEL
LIN {X 0,Y 278.555,Z 399.871,A -85,B 0,C 180,E1 -17425.412,E2 -17425.412} C_VEL
LIN {X 0,Y 277.662,Z 398.288,A -85,B 0,C 180,E1 -17426.162,E2 -17426.162} C_VEL
LIN {X 0,Y 277.242,Z 396.57,A -85,B 0,C 180,E1 -17426.901,E2 -17426.901} C_VEL
LIN {X 0,Y 277.225,Z 396.582,A -85,B 0,C 180,E1 -17431.206,E2 -17431.206} C_VEL
LIN {X 0,Y 277.221,Z 396.581,A -85,B 0,C 180,E1 -17434.471,E2 -17434.471} C_VEL
LIN {X 0,Y 277.235,Z 396.582,A -85,B 0,C 180,E1 -17437.651,E2 -17437.651} C_VEL
LIN {X 0,Y 277.258,Z 396.579,A -85,B 0,C 180,E1 -17440.76,E2 -17440.76} C_VEL
LIN {X 0,Y 277.356,Z 396.558,A -85,B 0,C 180,E1 -17445.322,E2 -17445.322} C_VEL
LIN {X 0,Y 277.442,Z 396.542,A -85,B 0,C 180,E1 -17449.787,E2 -17449.787} C_VEL
LIN {X 0,Y 277.587,Z 396.526,A -85,B 0,C 180,E1 -17452.728,E2 -17452.728} C_VEL
LIN {X 0,Y 277.794,Z 396.502,A -85,B 0,C 180,E1 -17458.551,E2 -17458.551} C_VEL
LIN {X 0,Y 277.801,Z 396.496,A -85,B 0,C 180,E1 -17461.45,E2 -17461.45} C_VEL
LIN {X 0,Y 277.585,Z 396.489,A -85,B 0,C 180,E1 -17467.273,E2 -17467.273} C_VEL
LIN {X 0,Y 277.445,Z 396.548,A -85,B 0,C 180,E1 -17470.214,E2 -17470.214} C_VEL
LIN {X 0,Y 277.4,Z 396.52,A -85,B 0,C 180,E1 -17474.676,E2 -17474.676} C_VEL
LIN {X 0,Y 277.315,Z 396.548,A -85,B 0,C 180,E1 -17479.236,E2 -17479.236} C_VEL
LIN {X 0,Y 277.252,Z 396.575,A -85,B 0,C 180,E1 -17483.928,E2 -17483.928} C_VEL
LIN {X 0,Y 277.233,Z 396.553,A -85,B 0,C 180,E1 -17487.472,E2 -17487.472} C_VEL
LIN {X 0,Y 277.241,Z 396.569,A -85,B 0,C 180,E1 -17490.474,E2 -17490.474} C_VEL
LIN {X 0,Y 277.235,Z 396.591,A -85,B 0,C 180,E1 -17493.698,E2 -17493.698} C_VEL
LIN {X 0,Y 278.02,Z 399.052,A -85,B 0,C 180,E1 -17494.007,E2 -17494.007} C_VEL
LIN {X 0,Y 279.977,Z 401.334,A -85,B 0,C 180,E1 -17494.607,E2 -17494.607} C_VEL
LIN {X 0,Y 280.989,Z 402.247,A -85,B 0,C 180,E1 -17494.9,E2 -17494.9} C_VEL
LIN {X 0,Y 283.033,Z 405.465,A -85,B 0,C 180,E1 -17495.534,E2 -17495.534} C_VEL
LIN {X 0,Y 284.723,Z 407.375,A -85,B 0,C 180,E1 -17496.015,E2 -17496.015} C_VEL
LIN {X 0,Y 287.471,Z 411.052,A -85,B 0,C 180,E1 -17496.797,E2 -17496.797} C_VEL
LIN {X 0,Y 296.827,Z 424.53,A -85,B 0,C 180,E1 -17499.299,E2 -17499.299} C_VEL
LIN {X 0,Y 305.536,Z 438.109,A -85,B 0,C 180,E1 -17501.428,E2 -17501.428} C_VEL
LIN {X 0,Y 313.88,Z 452.726,A -85,B 0,C 180,E1 -17503.339,E2 -17503.339} C_VEL
LIN {X 0,Y 314.575,Z 454.466,A -85,B 0,C 180,E1 -17503.506,E2 -17503.506} C_VEL
LIN {X 0,Y 312,Z 512.78,A -85,B 0,C 180,E1 -17504.843,E2 -17504.843} C_VEL
LIN {X 0,Y 311.311,Z 534.475,A -85,B 0,C 180,E1 -17505.464,E2 -17505.464} C_VEL
LIN {X 0,Y 310.291,Z 549.194,A -85,B 0,C 180,E1 -17506.123,E2 -17506.123} C_VEL
LIN {X 0,Y 308.796,Z 562.741,A -85,B 0,C 180,E1 -17506.941,E2 -17506.941} C_VEL
LIN {X 0,Y 306.992,Z 575.67,A -85,B 0,C 180,E1 -17507.964,E2 -17507.964} C_VEL
LIN {X 0,Y 304.528,Z 589.373,A -85,B 0,C 180,E1 -17509.312,E2 -17509.312} C_VEL
LIN {X 0,Y 301.927,Z 601.194,A -85,B 0,C 180,E1 -17510.74,E2 -17510.74} C_VEL
LIN {X 0,Y 298.907,Z 613.339,A -85,B 0,C 180,E1 -17512.529,E2 -17512.529} C_VEL
LIN {X 0,Y 295.956,Z 623.918,A -85,B 0,C 180,E1 -17514.425,E2 -17514.425} C_VEL
LIN {X 0,Y 292.935,Z 633.622,A -85,B 0,C 180,E1 -17516.51,E2 -17516.51} C_VEL
LIN {X 0,Y 289.787,Z 643.026,A -85,B 0,C 180,E1 -17518.98,E2 -17518.98} C_VEL
LIN {X 0,Y 286.911,Z 650.966,A -85,B 0,C 180,E1 -17521.549,E2 -17521.549} C_VEL
LIN {X 0,Y 284.249,Z 657.913,A -85,B 0,C 180,E1 -17524.363,E2 -17524.363} C_VEL
LIN {X 0,Y 282.177,Z 663.264,A -85,B 0,C 180,E1 -17527.153,E2 -17527.153} C_VEL
LIN {X 0,Y 280.734,Z 666.749,A -85,B 0,C 180,E1 -17529.484,E2 -17529.484} C_VEL
LIN {X 0,Y 279.352,Z 669.938,A -85,B 0,C 180,E1 -17532.429,E2 -17532.429} C_VEL
LIN {X 0,Y 278.375,Z 671.931,A -85,B 0,C 180,E1 -17535.378,E2 -17535.378} C_VEL
LIN {X 0,Y 277.883,Z 672.772,A -85,B 0,C 180,E1 -17538.328,E2 -17538.328} C_VEL
LIN {X 0,Y 277.717,Z 672.511,A -85,B 0,C 180,E1 -17541.267,E2 -17541.267} C_VEL
LIN {X 0,Y 277.693,Z 671.173,A -85,B 0,C 180,E1 -17544.19,E2 -17544.19} C_VEL
LIN {X 0,Y 278.066,Z 668.662,A -85,B 0,C 180,E1 -17547.103,E2 -17547.103} C_VEL
LIN {X 0,Y 278.854,Z 664.977,A -85,B 0,C 180,E1 -17550.001,E2 -17550.001} C_VEL
LIN {X 0,Y 279.884,Z 660.072,A -85,B 0,C 180,E1 -17552.879,E2 -17552.879} C_VEL
LIN {X 0,Y 281.377,Z 653.785,A -85,B 0,C 180,E1 -17555.734,E2 -17555.734} C_VEL
LIN {X 0,Y 283.165,Z 645.961,A -85,B 0,C 180,E1 -17558.564,E2 -17558.564} C_VEL
LIN {X 0,Y 285.154,Z 637.607,A -85,B 0,C 180,E1 -17561.012,E2 -17561.012} C_VEL
LIN {X 0,Y 287.478,Z 627.567,A -85,B 0,C 180,E1 -17563.43,E2 -17563.43} C_VEL
LIN {X 0,Y 289.643,Z 617.312,A -85,B 0,C 180,E1 -17565.48,E2 -17565.48} C_VEL
LIN {X 0,Y 291.695,Z 606.197,A -85,B 0,C 180,E1 -17567.347,E2 -17567.347} C_VEL
LIN {X 0,Y 293.83,Z 594.092,A -85,B 0,C 180,E1 -17569.02,E2 -17569.02} C_VEL
LIN {X 0,Y 295.856,Z 580.855,A -85,B 0,C 180,E1 -17570.511,E2 -17570.511} C_VEL
LIN {X 0,Y 297.662,Z 567.12,A -85,B 0,C 180,E1 -17571.74,E2 -17571.74} C_VEL
LIN {X 0,Y 299.152,Z 551.644,A -85,B 0,C 180,E1 -17572.807,E2 -17572.807} C_VEL
LIN {X 0,Y 300.124,Z 536.471,A -85,B 0,C 180,E1 -17573.568,E2 -17573.568} C_VEL
LIN {X 0,Y 300.604,Z 520.761,A -85,B 0,C 180,E1 -17574.085,E2 -17574.085} C_VEL
LIN {X 0,Y 302.884,Z 450.001,A -85,B 0,C 180,E1 -17575.762,E2 -17575.762} C_VEL
LIN {X 0,Y 303.002,Z 444.383,A -85,B 0,C 180,E1 -17575.903,E2 -17575.903} C_VEL
LIN {X 0,Y 295.132,Z 428.361,A -85,B 0,C 180,E1 -17577.339,E2 -17577.339} C_VEL
LIN {X 0,Y 285.844,Z 411.561,A -85,B 0,C 180,E1 -17579.101,E2 -17579.101} C_VEL
LIN {X 0,Y 278.998,Z 400.446,A -85,B 0,C 180,E1 -17580.459,E2 -17580.459} C_VEL
LIN {X 0,Y 277.449,Z 397.638,A -85,B 0,C 180,E1 -17580.789,E2 -17580.789} C_VEL
LIN {X 0,Y 277.243,Z 396.559,A -85,B 0,C 180,E1 -17580.891,E2 -17580.891} C_VEL
LIN {X 0,Y 277.246,Z 396.571,A -85,B 0,C 180,E1 -17583.895,E2 -17583.895} C_VEL
LIN {X 0,Y 277.248,Z 396.571,A -85,B 0,C 180,E1 -17587.472,E2 -17587.472} C_VEL
LIN {X 0,Y 277.172,Z 396.582,A -85,B 0,C 180,E1 -17591.243,E2 -17591.243} C_VEL
LIN {X 0,Y 277.172,Z 396.585,A -85,B 0,C 180,E1 -17595.232,E2 -17595.232} C_VEL
LIN {X 0,Y 277.174,Z 396.582,A -85,B 0,C 180,E1 -17598.756,E2 -17598.756} C_VEL
LIN {X 0,Y 277.23,Z 396.572,A -85,B 0,C 180,E1 -17602.524,E2 -17602.524} C_VEL
LIN {X 0,Y 277.243,Z 396.565,A -85,B 0,C 180,E1 -17606.103,E2 -17606.103} C_VEL
LIN {X 0,Y 277.226,Z 396.576,A -85,B 0,C 180,E1 -17609.534,E2 -17609.534} C_VEL
LIN {X 0,Y 277.192,Z 396.572,A -85,B 0,C 180,E1 -17610.708,E2 -17610.708} C_VEL
LIN {X 0,Y 276.562,Z 396.656,A -85,B 0,C 180,E1 -17611.921,E2 -17611.921} C_VEL
LIN {X 0,Y 273.765,Z 397.009,A -85,B 0,C 180,E1 -17613.897,E2 -17613.897} C_VEL
LIN {X 0,Y 271.355,Z 397.306,A -85,B 0,C 180,E1 -17615.502,E2 -17615.502} C_VEL
LIN {X 0,Y 270.289,Z 397.435,A -85,B 0,C 180,E1 -17616.746,E2 -17616.746} C_VEL
LIN {X 0,Y 270.186,Z 397.446,A -85,B 0,C 180,E1 -17617.167,E2 -17617.167} C_VEL
LIN {X 0,Y 270.22,Z 397.443,A -85,B 0,C 180,E1 -17620.238,E2 -17620.238} C_VEL
LIN {X 0,Y 270.364,Z 397.429,A -85,B 0,C 180,E1 -17624.933,E2 -17624.933} C_VEL
LIN {X 0,Y 270.382,Z 397.374,A -85,B 0,C 180,E1 -17629.516,E2 -17629.516} C_VEL
LIN {X 0,Y 270.546,Z 397.395,A -85,B 0,C 180,E1 -17632.537,E2 -17632.537} C_VEL
LIN {X 0,Y 270.76,Z 397.368,A -85,B 0,C 180,E1 -17638.512,E2 -17638.512} C_VEL
LIN {X 0,Y 270.764,Z 397.381,A -85,B 0,C 180,E1 -17641.487,E2 -17641.487} C_VEL
LIN {X 0,Y 270.554,Z 397.405,A -85,B 0,C 180,E1 -17647.462,E2 -17647.462} C_VEL
LIN {X 0,Y 270.38,Z 397.424,A -85,B 0,C 180,E1 -17650.483,E2 -17650.483} C_VEL
LIN {X 0,Y 270.332,Z 397.427,A -85,B 0,C 180,E1 -17655.068,E2 -17655.068} C_VEL
LIN {X 0,Y 270.212,Z 397.446,A -85,B 0,C 180,E1 -17659.762,E2 -17659.762} C_VEL
LIN {X 0,Y 270.179,Z 397.456,A -85,B 0,C 180,E1 -17664.437,E2 -17664.437} C_VEL
LIN {X 0,Y 270.18,Z 397.458,A -85,B 0,C 180,E1 -17667.919,E2 -17667.919} C_VEL
LIN {X 0,Y 270.165,Z 397.461,A -85,B 0,C 180,E1 -17671.35,E2 -17671.35} C_VEL
LIN {X 0,Y 270.193,Z 397.441,A -85,B 0,C 180,E1 -17674.906,E2 -17674.906} C_VEL
LIN {X 0,Y 270.195,Z 397.438,A -85,B 0,C 180,E1 -17678.711,E2 -17678.711} C_VEL
LIN {X 0,Y 270.163,Z 397.533,A -85,B 0,C 180,E1 -17680.017,E2 -17680.017} C_VEL
LIN {X 0,Y 274.21,Z 410.039,A -85,B 0,C 180,E1 -17683.789,E2 -17683.789} C_VEL
LIN {X 0,Y 276.926,Z 419.162,A -85,B 0,C 180,E1 -17686.33,E2 -17686.33} C_VEL
LIN {X 0,Y 280.354,Z 432.205,A -85,B 0,C 180,E1 -17689.66,E2 -17689.66} C_VEL
LIN {X 0,Y 287.9,Z 449.796,A -85,B 0,C 180,E1 -17691.254,E2 -17691.254} C_VEL
LIN {X 0,Y 291.015,Z 476.048,A -85,B 0,C 180,E1 -17692.43,E2 -17692.43} C_VEL
LIN {X 0,Y 295.272,Z 516.814,A -85,B 0,C 180,E1 -17694.112,E2 -17694.112} C_VEL
LIN {X 0,Y 291.979,Z 603.096,A -85,B 0,C 180,E1 -17696.178,E2 -17696.178} C_VEL
LIN {X 0,Y 290.68,Z 618.596,A -85,B 0,C 180,E1 -17696.786,E2 -17696.786} C_VEL
LIN {X 0,Y 288.857,Z 633.627,A -85,B 0,C 180,E1 -17697.638,E2 -17697.638} C_VEL
LIN {X 0,Y 286.476,Z 648.717,A -85,B 0,C 180,E1 -17698.785,E2 -17698.785} C_VEL
LIN {X 0,Y 283.874,Z 661.835,A -85,B 0,C 180,E1 -17700.055,E2 -17700.055} C_VEL
LIN {X 0,Y 281.206,Z 674.937,A -85,B 0,C 180,E1 -17701.65,E2 -17701.65} C_VEL
LIN {X 0,Y 278.705,Z 686.73,A -85,B 0,C 180,E1 -17703.411,E2 -17703.411} C_VEL
LIN {X 0,Y 276.014,Z 698.639,A -85,B 0,C 180,E1 -17705.558,E2 -17705.558} C_VEL
LIN {X 0,Y 273.821,Z 708.696,A -85,B 0,C 180,E1 -17707.754,E2 -17707.754} C_VEL
LIN {X 0,Y 271.881,Z 718.609,A -85,B 0,C 180,E1 -17710.364,E2 -17710.364} C_VEL
LIN {X 0,Y 270.445,Z 726.882,A -85,B 0,C 180,E1 -17713.001,E2 -17713.001} C_VEL
LIN {X 0,Y 269.617,Z 733.792,A -85,B 0,C 180,E1 -17715.662,E2 -17715.662} C_VEL
LIN {X 0,Y 269.178,Z 740.152,A -85,B 0,C 180,E1 -17718.707,E2 -17718.707} C_VEL
LIN {X 0,Y 269.269,Z 743.941,A -85,B 0,C 180,E1 -17720.99,E2 -17720.99} C_VEL
LIN {X 0,Y 269.645,Z 747.822,A -85,B 0,C 180,E1 -17724.015,E2 -17724.015} C_VEL
LIN {X 0,Y 269.833,Z 749.254,A -85,B 0,C 180,E1 -17725.518,E2 -17725.518} C_VEL
LIN {X 0,Y 270.286,Z 751.161,A -85,B 0,C 180,E1 -17728.509,E2 -17728.509} C_VEL
LIN {X 0,Y 270.553,Z 751.644,A -85,B 0,C 180,E1 -17729.999,E2 -17729.999} C_VEL
LIN {X 0,Y 270.245,Z 751.709,A -85,B 0,C 180,E1 -17731.49,E2 -17731.49} C_VEL
LIN {X 0,Y 269.729,Z 750.926,A -85,B 0,C 180,E1 -17734.483,E2 -17734.483} C_VEL
LIN {X 0,Y 269.199,Z 748.926,A -85,B 0,C 180,E1 -17737.5,E2 -17737.5} C_VEL
LIN {X 0,Y 268.959,Z 745.729,A -85,B 0,C 180,E1 -17740.539,E2 -17740.539} C_VEL
LIN {X 0,Y 269.257,Z 741.306,A -85,B 0,C 180,E1 -17743.586,E2 -17743.586} C_VEL
LIN {X 0,Y 270.26,Z 735.554,A -85,B 0,C 180,E1 -17746.621,E2 -17746.621} C_VEL
LIN {X 0,Y 271.997,Z 728.359,A -85,B 0,C 180,E1 -17749.626,E2 -17749.626} C_VEL
LIN {X 0,Y 274.461,Z 719.559,A -85,B 0,C 180,E1 -17752.587,E2 -17752.587} C_VEL
LIN {X 0,Y 277.367,Z 710.291,A -85,B 0,C 180,E1 -17755.112,E2 -17755.112} C_VEL
LIN {X 0,Y 280.792,Z 699.265,A -85,B 0,C 180,E1 -17757.582,E2 -17757.582} C_VEL
LIN {X 0,Y 284.67,Z 687.032,A -85,B 0,C 180,E1 -17759.79,E2 -17759.79} C_VEL
LIN {X 0,Y 288.375,Z 674.634,A -85,B 0,C 180,E1 -17761.597,E2 -17761.597} C_VEL
LIN {X 0,Y 292.091,Z 661.063,A -85,B 0,C 180,E1 -17763.186,E2 -17763.186} C_VEL
LIN {X 0,Y 295.402,Z 647.806,A -85,B 0,C 180,E1 -17764.404,E2 -17764.404} C_VEL
LIN {X 0,Y 298.446,Z 633.372,A -85,B 0,C 180,E1 -17765.441,E2 -17765.441} C_VEL
LIN {X 0,Y 300.858,Z 618.527,A -85,B 0,C 180,E1 -17766.247,E2 -17766.247} C_VEL
LIN {X 0,Y 302.462,Z 604.424,A -85,B 0,C 180,E1 -17766.8,E2 -17766.8} C_VEL
LIN {X 0,Y 303.68,Z 583.212,A -85,B 0,C 180,E1 -17767.354,E2 -17767.354} C_VEL
LIN {X 0,Y 306.607,Z 517.117,A -85,B 0,C 180,E1 -17768.899,E2 -17768.899} C_VEL
LIN {X 0,Y 304.589,Z 496.7,A -85,B 0,C 180,E1 -17769.875,E2 -17769.875} C_VEL
LIN {X 0,Y 301.62,Z 472.858,A -85,B 0,C 180,E1 -17771.164,E2 -17771.164} C_VEL
LIN {X 0,Y 300.188,Z 463.928,A -85,B 0,C 180,E1 -17771.72,E2 -17771.72} C_VEL
LIN {X 0,Y 293.357,Z 449.546,A -85,B 0,C 180,E1 -17773.542,E2 -17773.542} C_VEL
LIN {X 0,Y 287.5,Z 438.3,A -85,B 0,C 180,E1 -17775.188,E2 -17775.188} C_VEL
LIN {X 0,Y 283.594,Z 431.496,A -85,B 0,C 180,E1 -17776.33,E2 -17776.33} C_VEL
LIN {X 0,Y 280.518,Z 425.833,A -85,B 0,C 180,E1 -17777.336,E2 -17777.336} C_VEL
LIN {X 0,Y 277.298,Z 416.275,A -85,B 0,C 180,E1 -17780.683,E2 -17780.683} C_VEL
LIN {X 0,Y 274.298,Z 407.994,A -85,B 0,C 180,E1 -17783.893,E2 -17783.893} C_VEL
LIN {X 0,Y 272.253,Z 402.95,A -85,B 0,C 180,E1 -17786.067,E2 -17786.067} C_VEL
LIN {X 0,Y 270.172,Z 397.454,A -85,B 0,C 180,E1 -17788.651,E2 -17788.651} C_VEL
LIN {X 0,Y 270.182,Z 397.451,A -85,B 0,C 180,E1 -17792.175,E2 -17792.175} C_VEL
LIN {X 0,Y 270.172,Z 397.452,A -85,B 0,C 180,E1 -17795.564,E2 -17795.564} C_VEL
LIN {X 0,Y 270.205,Z 397.452,A -85,B 0,C 180,E1 -17800.237,E2 -17800.237} C_VEL
LIN {X 0,Y 270.327,Z 397.438,A -85,B 0,C 180,E1 -17804.931,E2 -17804.931} C_VEL
LIN {X 0,Y 270.374,Z 397.423,A -85,B 0,C 180,E1 -17809.517,E2 -17809.517} C_VEL
LIN {X 0,Y 270.55,Z 397.405,A -85,B 0,C 180,E1 -17812.537,E2 -17812.537} C_VEL
LIN {X 0,Y 270.759,Z 397.377,A -85,B 0,C 180,E1 -17818.513,E2 -17818.513} C_VEL
LIN {X 0,Y 270.765,Z 397.372,A -85,B 0,C 180,E1 -17821.488,E2 -17821.488} C_VEL
LIN {X 0,Y 270.545,Z 397.366,A -85,B 0,C 180,E1 -17827.463,E2 -17827.463} C_VEL
LIN {X 0,Y 270.399,Z 397.427,A -85,B 0,C 180,E1 -17830.483,E2 -17830.483} C_VEL
LIN {X 0,Y 270.368,Z 397.397,A -85,B 0,C 180,E1 -17835.067,E2 -17835.067} C_VEL
LIN {X 0,Y 270.252,Z 397.419,A -85,B 0,C 180,E1 -17839.76,E2 -17839.76} C_VEL
LIN {X 0,Y 270.171,Z 397.453,A -85,B 0,C 180,E1 -17844.596,E2 -17844.596} C_VEL
LIN {X 0,Y 270.181,Z 397.435,A -85,B 0,C 180,E1 -17847.919,E2 -17847.919} C_VEL
LIN {X 0,Y 270.176,Z 397.436,A -85,B 0,C 180,E1 -17851.732,E2 -17851.732} C_VEL
LIN {X 0,Y 271.117,Z 400.164,A -85,B 0,C 180,E1 -17852.156,E2 -17852.156} C_VEL
LIN {X 0,Y 273.108,Z 402.341,A -85,B 0,C 180,E1 -17852.816,E2 -17852.816} C_VEL
LIN {X 0,Y 273.994,Z 403.043,A -85,B 0,C 180,E1 -17853.091,E2 -17853.091} C_VEL
LIN {X 0,Y 276.006,Z 406.309,A -85,B 0,C 180,E1 -17853.775,E2 -17853.775} C_VEL
LIN {X 0,Y 277.893,Z 408.303,A -85,B 0,C 180,E1 -17854.353,E2 -17854.353} C_VEL
LIN {X 0,Y 280.563,Z 411.954,A -85,B 0,C 180,E1 -17855.18,E2 -17855.18} C_VEL
LIN {X 0,Y 285.419,Z 418.663,A -85,B 0,C 180,E1 -17856.609,E2 -17856.609} C_VEL
LIN {X 0,Y 293.263,Z 430.054,A -85,B 0,C 180,E1 -17858.757,E2 -17858.757} C_VEL
LIN {X 0,Y 301.67,Z 443.363,A -85,B 0,C 180,E1 -17860.882,E2 -17860.882} C_VEL
LIN {X 0,Y 309.179,Z 456.63,A -85,B 0,C 180,E1 -17862.662,E2 -17862.662} C_VEL
LIN {X 0,Y 306.537,Z 516.401,A -85,B 0,C 180,E1 -17864.067,E2 -17864.067} C_VEL
LIN {X 0,Y 305.775,Z 536.866,A -85,B 0,C 180,E1 -17864.68,E2 -17864.68} C_VEL
LIN {X 0,Y 304.736,Z 551.3,A -85,B 0,C 180,E1 -17865.366,E2 -17865.366} C_VEL
LIN {X 0,Y 303.199,Z 564.328,A -85,B 0,C 180,E1 -17866.175,E2 -17866.175} C_VEL
LIN {X 0,Y 300.982,Z 579.005,A -85,B 0,C 180,E1 -17867.38,E2 -17867.38} C_VEL
LIN {X 0,Y 298.424,Z 592.26,A -85,B 0,C 180,E1 -17868.747,E2 -17868.747} C_VEL
LIN {X 0,Y 295.596,Z 604.456,A -85,B 0,C 180,E1 -17870.287,E2 -17870.287} C_VEL
LIN {X 0,Y 292.354,Z 616.713,A -85,B 0,C 180,E1 -17872.196,E2 -17872.196} C_VEL
LIN {X 0,Y 289.025,Z 627.776,A -85,B 0,C 180,E1 -17874.298,E2 -17874.298} C_VEL
LIN {X 0,Y 285.86,Z 637.322,A -85,B 0,C 180,E1 -17876.501,E2 -17876.501} C_VEL
LIN {X 0,Y 282.702,Z 646.019,A -85,B 0,C 180,E1 -17878.948,E2 -17878.948} C_VEL
LIN {X 0,Y 279.904,Z 653.392,A -85,B 0,C 180,E1 -17881.508,E2 -17881.508} C_VEL
LIN {X 0,Y 277.156,Z 660.202,A -85,B 0,C 180,E1 -17884.465,E2 -17884.465} C_VEL
LIN {X 0,Y 274.924,Z 665.47,A -85,B 0,C 180,E1 -17887.454,E2 -17887.454} C_VEL
LIN {X 0,Y 273.206,Z 669.358,A -85,B 0,C 180,E1 -17890.464,E2 -17890.464} C_VEL
LIN {X 0,Y 271.956,Z 671.998,A -85,B 0,C 180,E1 -17893.486,E2 -17893.486} C_VEL
LIN {X 0,Y 271.143,Z 673.47,A -85,B 0,C 180,E1 -17896.511,E2 -17896.511} C_VEL
LIN {X 0,Y 270.76,Z 673.817,A -85,B 0,C 180,E1 -17899.532,E2 -17899.532} C_VEL
LIN {X 0,Y 270.73,Z 673.056,A -85,B 0,C 180,E1 -17902.543,E2 -17902.543} C_VEL
LIN {X 0,Y 270.803,Z 671.182,A -85,B 0,C 180,E1 -17905.535,E2 -17905.535} C_VEL
LIN {X 0,Y 271.35,Z 668.156,A -85,B 0,C 180,E1 -17908.516,E2 -17908.516} C_VEL
LIN {X 0,Y 272.241,Z 663.942,A -85,B 0,C 180,E1 -17911.48,E2 -17911.48} C_VEL
LIN {X 0,Y 273.559,Z 658.429,A -85,B 0,C 180,E1 -17914.421,E2 -17914.421} C_VEL
LIN {X 0,Y 275.309,Z 651.464,A -85,B 0,C 180,E1 -17917.334,E2 -17917.334} C_VEL
LIN {X 0,Y 277.103,Z 644.039,A -85,B 0,C 180,E1 -17919.858,E2 -17919.858} C_VEL
LIN {X 0,Y 279.296,Z 635.105,A -85,B 0,C 180,E1 -17922.35,E2 -17922.35} C_VEL
LIN {X 0,Y 281.426,Z 626.028,A -85,B 0,C 180,E1 -17924.462,E2 -17924.462} C_VEL
LIN {X 0,Y 283.73,Z 615.263,A -85,B 0,C 180,E1 -17926.55,E2 -17926.55} C_VEL
LIN {X 0,Y 286.111,Z 602.387,A -85,B 0,C 180,E1 -17928.623,E2 -17928.623} C_VEL
LIN {X 0,Y 288.497,Z 589.2,A -85,B 0,C 180,E1 -17930.313,E2 -17930.313} C_VEL
LIN {X 0,Y 290.386,Z 576.284,A -85,B 0,C 180,E1 -17931.659,E2 -17931.659} C_VEL
LIN {X 0,Y 292.096,Z 562.121,A -85,B 0,C 180,E1 -17932.829,E2 -17932.829} C_VEL
LIN {X 0,Y 293.389,Z 547.512,A -85,B 0,C 180,E1 -17933.749,E2 -17933.749} C_VEL
LIN {X 0,Y 294.19,Z 532.097,A -85,B 0,C 180,E1 -17934.447,E2 -17934.447} C_VEL
LIN {X 0,Y 295.034,Z 500.49,A -85,B 0,C 180,E1 -17935.296,E2 -17935.296} C_VEL
LIN {X 0,Y 296.965,Z 446.474,A -85,B 0,C 180,E1 -17936.586,E2 -17936.586} C_VEL
LIN {X 0,Y 287.358,Z 427.27,A -85,B 0,C 180,E1 -17938.414,E2 -17938.414} C_VEL
LIN {X 0,Y 278.218,Z 411.355,A -85,B 0,C 180,E1 -17940.234,E2 -17940.234} C_VEL
LIN {X 0,Y 272.08,Z 401.451,A -85,B 0,C 180,E1 -17941.524,E2 -17941.524} C_VEL
LIN {X 0,Y 270.484,Z 398.758,A -85,B 0,C 180,E1 -17941.876,E2 -17941.876} C_VEL
LIN {X 0,Y 270.216,Z 397.45,A -85,B 0,C 180,E1 -17942.005,E2 -17942.005} C_VEL
LIN {X 0,Y 270.218,Z 397.446,A -85,B 0,C 180,E1 -17946.266,E2 -17946.266} C_VEL
LIN {X 0,Y 270.127,Z 397.454,A -85,B 0,C 180,E1 -17950.574,E2 -17950.574} C_VEL
LIN {X 0,Y 270.127,Z 397.458,A -85,B 0,C 180,E1 -17954.625,E2 -17954.625} C_VEL
LIN {X 0,Y 270.148,Z 397.451,A -85,B 0,C 180,E1 -17957.437,E2 -17957.437} C_VEL
LIN {X 0,Y 270.15,Z 397.452,A -85,B 0,C 180,E1 -17961.364,E2 -17961.364} C_VEL
LIN {X 0,Y 270.195,Z 397.45,A -85,B 0,C 180,E1 -17965.093,E2 -17965.093} C_VEL
LIN {X 0,Y 270.169,Z 397.458,A -85,B 0,C 180,E1 -17969.141,E2 -17969.141} C_VEL
LIN {X 0,Y 270.185,Z 397.452,A -85,B 0,C 180,E1 -17972.176,E2 -17972.176} C_VEL
LIN {X 0,Y 270.224,Z 397.439,A -85,B 0,C 180,E1 -17975.542,E2 -17975.542} C_VEL
LIN {X 0,Y 270.186,Z 397.446,A -85,B 0,C 180,E1 -17977.167,E2 -17977.167} C_VEL
LIN {X 0,Y 269.472,Z 397.545,A -85,B 0,C 180,E1 -17978.412,E2 -17978.412} C_VEL
LIN {X 0,Y 266.611,Z 397.891,A -85,B 0,C 180,E1 -17980.441,E2 -17980.441} C_VEL
LIN {X 0,Y 264.252,Z 398.186,A -85,B 0,C 180,E1 -17982.091,E2 -17982.091} C_VEL
LIN {X 0,Y 263.3,Z 398.312,A -85,B 0,C 180,E1 -17983.369,E2 -17983.369} C_VEL
LIN {X 0,Y 263.252,Z 398.317,A -85,B 0,C 180,E1 -17983.801,E2 -17983.801} C_VEL
LIN {X 0,Y 263.307,Z 398.266,A -85,B 0,C 180,E1 -17987.67,E2 -17987.67} C_VEL
LIN {X 0,Y 263.449,Z 398.248,A -85,B 0,C 180,E1 -17990.789,E2 -17990.789} C_VEL
LIN {X 0,Y 263.471,Z 398.29,A -85,B 0,C 180,E1 -17993.875,E2 -17993.875} C_VEL
LIN {X 0,Y 263.722,Z 398.244,A -85,B 0,C 180,E1 -17998.473,E2 -17998.473} C_VEL
LIN {X 0,Y 263.728,Z 398.257,A -85,B 0,C 180,E1 -18001.527,E2 -18001.527} C_VEL
LIN {X 0,Y 263.518,Z 398.279,A -85,B 0,C 180,E1 -18007.663,E2 -18007.663} C_VEL
LIN {X 0,Y 263.324,Z 398.305,A -85,B 0,C 180,E1 -18010.767,E2 -18010.767} C_VEL
LIN {X 0,Y 263.284,Z 398.308,A -85,B 0,C 180,E1 -18015.482,E2 -18015.482} C_VEL
LIN {X 0,Y 263.202,Z 398.325,A -85,B 0,C 180,E1 -18020.311,E2 -18020.311} C_VEL
LIN {X 0,Y 263.116,Z 398.335,A -85,B 0,C 180,E1 -18025.3,E2 -18025.3} C_VEL
LIN {X 0,Y 263.113,Z 398.335,A -85,B 0,C 180,E1 -18028.737,E2 -18028.737} C_VEL
LIN {X 0,Y 263.122,Z 398.326,A -85,B 0,C 180,E1 -18032.289,E2 -18032.289} C_VEL
LIN {X 0,Y 263.151,Z 398.334,A -85,B 0,C 180,E1 -18035.983,E2 -18035.983} C_VEL
LIN {X 0,Y 263.138,Z 398.351,A -85,B 0,C 180,E1 -18038.983,E2 -18038.983} C_VEL
LIN {X 0,Y 267.401,Z 411.449,A -85,B 0,C 180,E1 -18043.105,E2 -18043.105} C_VEL
LIN {X 0,Y 270.95,Z 423.598,A -85,B 0,C 180,E1 -18046.574,E2 -18046.574} C_VEL
LIN {X 0,Y 272.82,Z 430.865,A -85,B 0,C 180,E1 -18048.475,E2 -18048.475} C_VEL
LIN {X 0,Y 279.911,Z 446.811,A -85,B 0,C 180,E1 -18050.047,E2 -18050.047} C_VEL
LIN {X 0,Y 282.312,Z 452.975,A -85,B 0,C 180,E1 -18050.579,E2 -18050.579} C_VEL
LIN {X 0,Y 285.807,Z 483.546,A -85,B 0,C 180,E1 -18051.973,E2 -18051.973} C_VEL
LIN {X 0,Y 289.217,Z 516.975,A -85,B 0,C 180,E1 -18053.384,E2 -18053.384} C_VEL
LIN {X 0,Y 285.885,Z 602.069,A -85,B 0,C 180,E1 -18055.462,E2 -18055.462} C_VEL
LIN {X 0,Y 284.536,Z 617.578,A -85,B 0,C 180,E1 -18056.079,E2 -18056.079} C_VEL
LIN {X 0,Y 282.677,Z 632.623,A -85,B 0,C 180,E1 -18056.947,E2 -18056.947} C_VEL
LIN {X 0,Y 280.365,Z 646.714,A -85,B 0,C 180,E1 -18058.025,E2 -18058.025} C_VEL
LIN {X 0,Y 277.816,Z 659.514,A -85,B 0,C 180,E1 -18059.265,E2 -18059.265} C_VEL
LIN {X 0,Y 275.852,Z 668.663,A -85,B 0,C 180,E1 -18060.323,E2 -18060.323} C_VEL
LIN {X 0,Y 273.09,Z 681.876,A -85,B 0,C 180,E1 -18062.196,E2 -18062.196} C_VEL
LIN {X 0,Y 270.336,Z 693.443,A -85,B 0,C 180,E1 -18064.186,E2 -18064.186} C_VEL
LIN {X 0,Y 267.887,Z 704.124,A -85,B 0,C 180,E1 -18066.417,E2 -18066.417} C_VEL
LIN {X 0,Y 265.599,Z 714.622,A -85,B 0,C 180,E1 -18069.07,E2 -18069.07} C_VEL
LIN {X 0,Y 263.945,Z 723.379,A -85,B 0,C 180,E1 -18071.768,E2 -18071.768} C_VEL
LIN {X 0,Y 262.844,Z 730.675,A -85,B 0,C 180,E1 -18074.491,E2 -18074.491} C_VEL
LIN {X 0,Y 262.175,Z 737.462,A -85,B 0,C 180,E1 -18077.616,E2 -18077.616} C_VEL
LIN {X 0,Y 262.197,Z 742.78,A -85,B 0,C 180,E1 -18080.745,E2 -18080.745} C_VEL
LIN {X 0,Y 262.574,Z 746.71,A -85,B 0,C 180,E1 -18083.854,E2 -18083.854} C_VEL
LIN {X 0,Y 262.784,Z 748.167,A -85,B 0,C 180,E1 -18085.398,E2 -18085.398} C_VEL
LIN {X 0,Y 263.252,Z 750.116,A -85,B 0,C 180,E1 -18088.47,E2 -18088.47} C_VEL
LIN {X 0,Y 263.528,Z 750.606,A -85,B 0,C 180,E1 -18089.999,E2 -18089.999} C_VEL
LIN {X 0,Y 263.208,Z 750.681,A -85,B 0,C 180,E1 -18091.529,E2 -18091.529} C_VEL
LIN {X 0,Y 262.672,Z 749.931,A -85,B 0,C 180,E1 -18094.603,E2 -18094.603} C_VEL
LIN {X 0,Y 262.114,Z 747.959,A -85,B 0,C 180,E1 -18097.704,E2 -18097.704} C_VEL
LIN {X 0,Y 261.881,Z 744.794,A -85,B 0,C 180,E1 -18100.827,E2 -18100.827} C_VEL
LIN {X 0,Y 262.249,Z 740.406,A -85,B 0,C 180,E1 -18103.956,E2 -18103.956} C_VEL
LIN {X 0,Y 263.352,Z 734.68,A -85,B 0,C 180,E1 -18107.07,E2 -18107.07} C_VEL
LIN {X 0,Y 265.225,Z 727.534,A -85,B 0,C 180,E1 -18110.149,E2 -18110.149} C_VEL
LIN {X 0,Y 267.839,Z 718.791,A -85,B 0,C 180,E1 -18113.177,E2 -18113.177} C_VEL
LIN {X 0,Y 270.857,Z 709.584,A -85,B 0,C 180,E1 -18115.76,E2 -18115.76} C_VEL
LIN {X 0,Y 273.899,Z 700.296,A -85,B 0,C 180,E1 -18117.921,E2 -18117.921} C_VEL
LIN {X 0,Y 277.581,Z 689.461,A -85,B 0,C 180,E1 -18120.001,E2 -18120.001} C_VEL
LIN {X 0,Y 281.546,Z 676.79,A -85,B 0,C 180,E1 -18121.992,E2 -18121.992} C_VEL
LIN {X 0,Y 285.35,Z 663.612,A -85,B 0,C 180,E1 -18123.651,E2 -18123.651} C_VEL
LIN {X 0,Y 289.151,Z 649.427,A -85,B 0,C 180,E1 -18125.043,E2 -18125.043} C_VEL
LIN {X 0,Y 292.248,Z 635.725,A -85,B 0,C 180,E1 -18126.097,E2 -18126.097} C_VEL
LIN {X 0,Y 294.851,Z 621.303,A -85,B 0,C 180,E1 -18126.948,E2 -18126.948} C_VEL
LIN {X 0,Y 296.695,Z 606.823,A -85,B 0,C 180,E1 -18127.584,E2 -18127.584} C_VEL
LIN {X 0,Y 297.873,Z 591.67,A -85,B 0,C 180,E1 -18128.031,E2 -18128.031} C_VEL
LIN {X 0,Y 301.3,Z 518.264,A -85,B 0,C 180,E1 -18129.763,E2 -18129.763} C_VEL
LIN {X 0,Y 299.429,Z 498.581,A -85,B 0,C 180,E1 -18130.726,E2 -18130.726} C_VEL
LIN {X 0,Y 296.316,Z 472.535,A -85,B 0,C 180,E1 -18132.167,E2 -18132.167} C_VEL
LIN {X 0,Y 295.317,Z 467.025,A -85,B 0,C 180,E1 -18132.548,E2 -18132.548} C_VEL
LIN {X 0,Y 288.787,Z 453.271,A -85,B 0,C 180,E1 -18134.364,E2 -18134.364} C_VEL
LIN {X 0,Y 283.631,Z 443.205,A -85,B 0,C 180,E1 -18135.878,E2 -18135.878} C_VEL
LIN {X 0,Y 279.831,Z 436.45,A -85,B 0,C 180,E1 -18137.034,E2 -18137.034} C_VEL
LIN {X 0,Y 276.159,Z 430.06,A -85,B 0,C 180,E1 -18138.207,E2 -18138.207} C_VEL
LIN {X 0,Y 272.749,Z 424.128,A -85,B 0,C 180,E1 -18139.382,E2 -18139.382} C_VEL
LIN {X 0,Y 270.089,Z 416.332,A -85,B 0,C 180,E1 -18142.303,E2 -18142.303} C_VEL
LIN {X 0,Y 266.961,Z 407.908,A -85,B 0,C 180,E1 -18145.835,E2 -18145.835} C_VEL
LIN {X 0,Y 264.198,Z 401.271,A -85,B 0,C 180,E1 -18149.002,E2 -18149.002} C_VEL
LIN {X 0,Y 263.124,Z 398.334,A -85,B 0,C 180,E1 -18150.498,E2 -18150.498} C_VEL
LIN {X 0,Y 263.111,Z 398.336,A -85,B 0,C 180,E1 -18154.699,E2 -18154.699} C_VEL
LIN {X 0,Y 263.196,Z 398.321,A -85,B 0,C 180,E1 -18159.688,E2 -18159.688} C_VEL
LIN {X 0,Y 263.279,Z 398.318,A -85,B 0,C 180,E1 -18164.518,E2 -18164.518} C_VEL
LIN {X 0,Y 263.319,Z 398.303,A -85,B 0,C 180,E1 -18169.232,E2 -18169.232} C_VEL
LIN {X 0,Y 263.514,Z 398.283,A -85,B 0,C 180,E1 -18172.337,E2 -18172.337} C_VEL
LIN {X 0,Y 263.723,Z 398.253,A -85,B 0,C 180,E1 -18178.473,E2 -18178.473} C_VEL
LIN {X 0,Y 263.728,Z 398.248,A -85,B 0,C 180,E1 -18181.527,E2 -18181.527} C_VEL
LIN {X 0,Y 263.507,Z 398.242,A -85,B 0,C 180,E1 -18187.664,E2 -18187.664} C_VEL
LIN {X 0,Y 263.339,Z 398.309,A -85,B 0,C 180,E1 -18190.767,E2 -18190.767} C_VEL
LIN {X 0,Y 263.314,Z 398.278,A -85,B 0,C 180,E1 -18195.481,E2 -18195.481} C_VEL
LIN {X 0,Y 263.229,Z 398.289,A -85,B 0,C 180,E1 -18200.31,E2 -18200.31} C_VEL
LIN {X 0,Y 263.114,Z 398.319,A -85,B 0,C 180,E1 -18205.301,E2 -18205.301} C_VEL
LIN {X 0,Y 263.119,Z 398.34,A -85,B 0,C 180,E1 -18209.614,E2 -18209.614} C_VEL
LIN {X 0,Y 263.949,Z 400.866,A -85,B 0,C 180,E1 -18210.006,E2 -18210.006} C_VEL
LIN {X 0,Y 265.834,Z 403.067,A -85,B 0,C 180,E1 -18210.706,E2 -18210.706} C_VEL
LIN {X 0,Y 267.184,Z 404.105,A -85,B 0,C 180,E1 -18211.169,E2 -18211.169} C_VEL
LIN {X 0,Y 269.195,Z 407.356,A -85,B 0,C 180,E1 -18211.917,E2 -18211.917} C_VEL
LIN {X 0,Y 271.196,Z 409.44,A -85,B 0,C 180,E1 -18212.585,E2 -18212.585} C_VEL
LIN {X 0,Y 273.561,Z 412.77,A -85,B 0,C 180,E1 -18213.386,E2 -18213.386} C_VEL
LIN {X 0,Y 275.019,Z 414.517,A -85,B 0,C 180,E1 -18213.853,E2 -18213.853} C_VEL
LIN {X 0,Y 278.839,Z 419.716,A -85,B 0,C 180,E1 -18215.057,E2 -18215.057} C_VEL
LIN {X 0,Y 284.828,Z 428.267,A -85,B 0,C 180,E1 -18216.836,E2 -18216.836} C_VEL
LIN {X 0,Y 291.834,Z 438.81,A -85,B 0,C 180,E1 -18218.766,E2 -18218.766} C_VEL
LIN {X 0,Y 300.451,Z 453.076,A -85,B 0,C 180,E1 -18220.973,E2 -18220.973} C_VEL
LIN {X 0,Y 303.944,Z 459.535,A -85,B 0,C 180,E1 -18221.829,E2 -18221.829} C_VEL
LIN {X 0,Y 301.439,Z 511.59,A -85,B 0,C 180,E1 -18223.049,E2 -18223.049} C_VEL
LIN {X 0,Y 300.603,Z 535.551,A -85,B 0,C 180,E1 -18223.735,E2 -18223.735} C_VEL
LIN {X 0,Y 299.477,Z 550.685,A -85,B 0,C 180,E1 -18224.418,E2 -18224.418} C_VEL
LIN {X 0,Y 297.928,Z 563.958,A -85,B 0,C 180,E1 -18225.231,E2 -18225.231} C_VEL
LIN {X 0,Y 295.684,Z 578.689,A -85,B 0,C 180,E1 -18226.428,E2 -18226.428} C_VEL
LIN {X 0,Y 293.01,Z 592.197,A -85,B 0,C 180,E1 -18227.812,E2 -18227.812} C_VEL
LIN {X 0,Y 290.069,Z 604.54,A -85,B 0,C 180,E1 -18229.374,E2 -18229.374} C_VEL
LIN {X 0,Y 286.643,Z 616.98,A -85,B 0,C 180,E1 -18231.305,E2 -18231.305} C_VEL
LIN {X 0,Y 283.173,Z 628.169,A -85,B 0,C 180,E1 -18233.443,E2 -18233.443} C_VEL
LIN {X 0,Y 279.848,Z 637.794,A -85,B 0,C 180,E1 -18235.683,E2 -18235.683} C_VEL
LIN {X 0,Y 276.572,Z 646.582,A -85,B 0,C 180,E1 -18238.18,E2 -18238.18} C_VEL
LIN {X 0,Y 273.462,Z 654.351,A -85,B 0,C 180,E1 -18240.905,E2 -18240.905} C_VEL
LIN {X 0,Y 270.657,Z 660.932,A -85,B 0,C 180,E1 -18243.806,E2 -18243.806} C_VEL
LIN {X 0,Y 268.303,Z 666.267,A -85,B 0,C 180,E1 -18246.865,E2 -18246.865} C_VEL
LIN {X 0,Y 266.451,Z 670.222,A -85,B 0,C 180,E1 -18249.948,E2 -18249.948} C_VEL
LIN {X 0,Y 265.096,Z 672.922,A -85,B 0,C 180,E1 -18253.046,E2 -18253.046} C_VEL
LIN {X 0,Y 264.182,Z 674.455,A -85,B 0,C 180,E1 -18256.148,E2 -18256.148} C_VEL
LIN {X 0,Y 263.764,Z 674.857,A -85,B 0,C 180,E1 -18259.251,E2 -18259.251} C_VEL
LIN {X 0,Y 263.686,Z 674.126,A -85,B 0,C 180,E1 -18262.343,E2 -18262.343} C_VEL
LIN {X 0,Y 263.753,Z 672.305,A -85,B 0,C 180,E1 -18265.416,E2 -18265.416} C_VEL
LIN {X 0,Y 264.305,Z 669.339,A -85,B 0,C 180,E1 -18268.477,E2 -18268.477} C_VEL
LIN {X 0,Y 265.229,Z 665.184,A -85,B 0,C 180,E1 -18271.519,E2 -18271.519} C_VEL
LIN {X 0,Y 266.593,Z 659.735,A -85,B 0,C 180,E1 -18274.537,E2 -18274.537} C_VEL
LIN {X 0,Y 268.375,Z 652.845,A -85,B 0,C 180,E1 -18277.524,E2 -18277.524} C_VEL
LIN {X 0,Y 270.227,Z 645.501,A -85,B 0,C 180,E1 -18280.111,E2 -18280.111} C_VEL
LIN {X 0,Y 272.503,Z 636.656,A -85,B 0,C 180,E1 -18282.663,E2 -18282.663} C_VEL
LIN {X 0,Y 275.079,Z 625.991,A -85,B 0,C 180,E1 -18285.182,E2 -18285.182} C_VEL
LIN {X 0,Y 277.493,Z 615.059,A -85,B 0,C 180,E1 -18287.313,E2 -18287.313} C_VEL
LIN {X 0,Y 279.775,Z 603.102,A -85,B 0,C 180,E1 -18289.251,E2 -18289.251} C_VEL
LIN {X 0,Y 282.263,Z 589.842,A -85,B 0,C 180,E1 -18290.973,E2 -18290.973} C_VEL
LIN {X 0,Y 284.213,Z 576.878,A -85,B 0,C 180,E1 -18292.346,E2 -18292.346} C_VEL
LIN {X 0,Y 285.979,Z 562.607,A -85,B 0,C 180,E1 -18293.537,E2 -18293.537} C_VEL
LIN {X 0,Y 287.392,Z 547.05,A -85,B 0,C 180,E1 -18294.517,E2 -18294.517} C_VEL
LIN {X 0,Y 288.168,Z 531.543,A -85,B 0,C 180,E1 -18295.206,E2 -18295.206} C_VEL
LIN {X 0,Y 289.37,Z 491.374,A -85,B 0,C 180,E1 -18296.258,E2 -18296.258} C_VEL
LIN {X 0,Y 290.903,Z 448.477,A -85,B 0,C 180,E1 -18297.308,E2 -18297.308} C_VEL
LIN {X 0,Y 281.151,Z 429.157,A -85,B 0,C 180,E1 -18299.24,E2 -18299.24} C_VEL
LIN {X 0,Y 271.845,Z 413.121,A -85,B 0,C 180,E1 -18301.18,E2 -18301.18} C_VEL
LIN {X 0,Y 266.97,Z 405.415,A -85,B 0,C 180,E1 -18302.245,E2 -18302.245} C_VEL
LIN {X 0,Y 265.241,Z 402.533,A -85,B 0,C 180,E1 -18302.641,E2 -18302.641} C_VEL
LIN {X 0,Y 263.539,Z 399.902,A -85,B 0,C 180,E1 -18303.031,E2 -18303.031} C_VEL
LIN {X 0,Y 263.171,Z 398.326,A -85,B 0,C 180,E1 -18303.202,E2 -18303.202} C_VEL
LIN {X 0,Y 263.173,Z 398.322,A -85,B 0,C 180,E1 -18306.76,E2 -18306.76} C_VEL
LIN {X 0,Y 263.071,Z 398.332,A -85,B 0,C 180,E1 -18309.878,E2 -18309.878} C_VEL
LIN {X 0,Y 263.075,Z 398.332,A -85,B 0,C 180,E1 -18313.994,E2 -18313.994} C_VEL
LIN {X 0,Y 263.073,Z 398.334,A -85,B 0,C 180,E1 -18318.096,E2 -18318.096} C_VEL
LIN {X 0,Y 263.102,Z 398.329,A -85,B 0,C 180,E1 -18322.093,E2 -18322.093} C_VEL
LIN {X 0,Y 263.15,Z 398.321,A -85,B 0,C 180,E1 -18325.885,E2 -18325.885} C_VEL
LIN {X 0,Y 263.106,Z 398.334,A -85,B 0,C 180,E1 -18329.501,E2 -18329.501} C_VEL
LIN {X 0,Y 263.113,Z 398.336,A -85,B 0,C 180,E1 -18332.993,E2 -18332.993} C_VEL
LIN {X 0,Y 263.14,Z 398.321,A -85,B 0,C 180,E1 -18336.382,E2 -18336.382} C_VEL
LIN {X 0,Y 263.206,Z 398.319,A -85,B 0,C 180,E1 -18339.688,E2 -18339.688} C_VEL
LIN {X 0,Y 263.252,Z 398.317,A -85,B 0,C 180,E1 -18343.801,E2 -18343.801} C_VEL
LIN {X 0,Y 262.673,Z 398.388,A -85,B 0,C 180,E1 -18345.077,E2 -18345.077} C_VEL
LIN {X 0,Y 259.89,Z 398.707,A -85,B 0,C 180,E1 -18347.159,E2 -18347.159} C_VEL
LIN {X 0,Y 257.489,Z 398.983,A -85,B 0,C 180,E1 -18348.852,E2 -18348.852} C_VEL
LIN {X 0,Y 256.471,Z 399.108,A -85,B 0,C 180,E1 -18350.165,E2 -18350.165} C_VEL
LIN {X 0,Y 256.396,Z 399.122,A -85,B 0,C 180,E1 -18350.609,E2 -18350.609} C_VEL
LIN {X 0,Y 256.443,Z 399.163,A -85,B 0,C 180,E1 -18353.706,E2 -18353.706} C_VEL
LIN {X 0,Y 256.683,Z 399.12,A -85,B 0,C 180,E1 -18358.431,E2 -18358.431} C_VEL
LIN {X 0,Y 256.69,Z 399.133,A -85,B 0,C 180,E1 -18361.569,E2 -18361.569} C_VEL
LIN {X 0,Y 256.446,Z 399.164,A -85,B 0,C 180,E1 -18366.293,E2 -18366.293} C_VEL
LIN {X 0,Y 256.398,Z 399.157,A -85,B 0,C 180,E1 -18369.466,E2 -18369.466} C_VEL
LIN {X 0,Y 256.192,Z 399.185,A -85,B 0,C 180,E1 -18374.293,E2 -18374.293} C_VEL
LIN {X 0,Y 256.138,Z 399.202,A -85,B 0,C 180,E1 -18377.567,E2 -18377.567} C_VEL
LIN {X 0,Y 256.114,Z 399.209,A -85,B 0,C 180,E1 -18381.096,E2 -18381.096} C_VEL
LIN {X 0,Y 256.079,Z 399.213,A -85,B 0,C 180,E1 -18385.088,E2 -18385.088} C_VEL
LIN {X 0,Y 256.072,Z 399.212,A -85,B 0,C 180,E1 -18388.569,E2 -18388.569} C_VEL
LIN {X 0,Y 256.066,Z 399.212,A -85,B 0,C 180,E1 -18391.699,E2 -18391.699} C_VEL
LIN {X 0,Y 256.075,Z 399.202,A -85,B 0,C 180,E1 -18395.194,E2 -18395.194} C_VEL
LIN {X 0,Y 256.111,Z 399.363,A -85,B 0,C 180,E1 -18397.94,E2 -18397.94} C_VEL
LIN {X 0,Y 259.664,Z 410.177,A -85,B 0,C 180,E1 -18401.537,E2 -18401.537} C_VEL
LIN {X 0,Y 263.208,Z 421.68,A -85,B 0,C 180,E1 -18405.038,E2 -18405.038} C_VEL
LIN {X 0,Y 265.393,Z 429.631,A -85,B 0,C 180,E1 -18407.225,E2 -18407.225} C_VEL
LIN {X 0,Y 272.973,Z 446.371,A -85,B 0,C 180,E1 -18408.997,E2 -18408.997} C_VEL
LIN {X 0,Y 276.663,Z 455.606,A -85,B 0,C 180,E1 -18409.846,E2 -18409.846} C_VEL
LIN {X 0,Y 279.919,Z 484.848,A -85,B 0,C 180,E1 -18411.214,E2 -18411.214} C_VEL
LIN {X 0,Y 283.167,Z 517.09,A -85,B 0,C 180,E1 -18412.62,E2 -18412.62} C_VEL
LIN {X 0,Y 279.8,Z 600.996,A -85,B 0,C 180,E1 -18414.711,E2 -18414.711} C_VEL
LIN {X 0,Y 278.408,Z 616.525,A -85,B 0,C 180,E1 -18415.336,E2 -18415.336} C_VEL
LIN {X 0,Y 276.523,Z 631.592,A -85,B 0,C 180,E1 -18416.223,E2 -18416.223} C_VEL
LIN {X 0,Y 273.947,Z 646.674,A -85,B 0,C 180,E1 -18417.402,E2 -18417.402} C_VEL
LIN {X 0,Y 271.122,Z 660.287,A -85,B 0,C 180,E1 -18418.773,E2 -18418.773} C_VEL
LIN {X 0,Y 269.03,Z 669.648,A -85,B 0,C 180,E1 -18419.928,E2 -18419.928} C_VEL
LIN {X 0,Y 266.194,Z 682.501,A -85,B 0,C 180,E1 -18421.84,E2 -18421.84} C_VEL
LIN {X 0,Y 263.382,Z 693.833,A -85,B 0,C 180,E1 -18423.878,E2 -18423.878} C_VEL
LIN {X 0,Y 260.885,Z 704.34,A -85,B 0,C 180,E1 -18426.166,E2 -18426.166} C_VEL
LIN {X 0,Y 258.555,Z 714.626,A -85,B 0,C 180,E1 -18428.89,E2 -18428.89} C_VEL
LIN {X 0,Y 256.886,Z 723.235,A -85,B 0,C 180,E1 -18431.662,E2 -18431.662} C_VEL
LIN {X 0,Y 255.656,Z 731.315,A -85,B 0,C 180,E1 -18434.861,E2 -18434.861} C_VEL
LIN {X 0,Y 255.066,Z 737.762,A -85,B 0,C 180,E1 -18438.073,E2 -18438.073} C_VEL
LIN {X 0,Y 255.2,Z 742.765,A -85,B 0,C 180,E1 -18441.288,E2 -18441.288} C_VEL
LIN {X 0,Y 255.484,Z 745.593,A -85,B 0,C 180,E1 -18443.682,E2 -18443.682} C_VEL
LIN {X 0,Y 255.733,Z 747.079,A -85,B 0,C 180,E1 -18445.27,E2 -18445.27} C_VEL
LIN {X 0,Y 256.216,Z 749.064,A -85,B 0,C 180,E1 -18448.428,E2 -18448.428} C_VEL
LIN {X 0,Y 256.502,Z 749.563,A -85,B 0,C 180,E1 -18449.999,E2 -18449.999} C_VEL
LIN {X 0,Y 256.171,Z 749.654,A -85,B 0,C 180,E1 -18451.571,E2 -18451.571} C_VEL
LIN {X 0,Y 255.593,Z 748.932,A -85,B 0,C 180,E1 -18454.731,E2 -18454.731} C_VEL
LIN {X 0,Y 255.024,Z 746.991,A -85,B 0,C 180,E1 -18457.919,E2 -18457.919} C_VEL
LIN {X 0,Y 254.819,Z 743.86,A -85,B 0,C 180,E1 -18461.131,E2 -18461.131} C_VEL
LIN {X 0,Y 255.258,Z 739.497,A -85,B 0,C 180,E1 -18464.346,E2 -18464.346} C_VEL
LIN {X 0,Y 256.467,Z 733.811,A -85,B 0,C 180,E1 -18467.543,E2 -18467.543} C_VEL
LIN {X 0,Y 258.486,Z 726.717,A -85,B 0,C 180,E1 -18470.698,E2 -18470.698} C_VEL
LIN {X 0,Y 261.251,Z 718.027,A -85,B 0,C 180,E1 -18473.797,E2 -18473.797} C_VEL
LIN {X 0,Y 264.371,Z 708.876,A -85,B 0,C 180,E1 -18476.44,E2 -18476.44} C_VEL
LIN {X 0,Y 267.566,Z 699.659,A -85,B 0,C 180,E1 -18478.642,E2 -18478.642} C_VEL
LIN {X 0,Y 271.383,Z 688.906,A -85,B 0,C 180,E1 -18480.76,E2 -18480.76} C_VEL
LIN {X 0,Y 275.228,Z 677.286,A -85,B 0,C 180,E1 -18482.643,E2 -18482.643} C_VEL
LIN {X 0,Y 279.046,Z 664.732,A -85,B 0,C 180,E1 -18484.299,E2 -18484.299} C_VEL
LIN {X 0,Y 282.933,Z 651.061,A -85,B 0,C 180,E1 -18485.712,E2 -18485.712} C_VEL
LIN {X 0,Y 286.332,Z 636.961,A -85,B 0,C 180,E1 -18486.855,E2 -18486.855} C_VEL
LIN {X 0,Y 289.122,Z 622.516,A -85,B 0,C 180,E1 -18487.751,E2 -18487.751} C_VEL
LIN {X 0,Y 291.241,Z 606.934,A -85,B 0,C 180,E1 -18488.47,E2 -18488.47} C_VEL
LIN {X 0,Y 292.541,Z 591.431,A -85,B 0,C 180,E1 -18488.941,E2 -18488.941} C_VEL
LIN {X 0,Y 296.052,Z 520.027,A -85,B 0,C 180,E1 -18490.64,E2 -18490.64} C_VEL
LIN {X 0,Y 294.652,Z 503.274,A -85,B 0,C 180,E1 -18491.454,E2 -18491.454} C_VEL
LIN {X 0,Y 291.356,Z 474.566,A -85,B 0,C 180,E1 -18493.077,E2 -18493.077} C_VEL
LIN {X 0,Y 290.508,Z 470.125,A -85,B 0,C 180,E1 -18493.405,E2 -18493.405} C_VEL
LIN {X 0,Y 284.16,Z 456.691,A -85,B 0,C 180,E1 -18495.252,E2 -18495.252} C_VEL
LIN {X 0,Y 279.114,Z 446.853,A -85,B 0,C 180,E1 -18496.801,E2 -18496.801} C_VEL
LIN {X 0,Y 276.254,Z 441.592,A -85,B 0,C 180,E1 -18497.715,E2 -18497.715} C_VEL
LIN {X 0,Y 272.489,Z 434.998,A -85,B 0,C 180,E1 -18498.965,E2 -18498.965} C_VEL
LIN {X 0,Y 268.653,Z 428.565,A -85,B 0,C 180,E1 -18500.301,E2 -18500.301} C_VEL
LIN {X 0,Y 264.807,Z 422.028,A -85,B 0,C 180,E1 -18501.778,E2 -18501.778} C_VEL
LIN {X 0,Y 261.505,Z 412.842,A -85,B 0,C 180,E1 -18505.641,E2 -18505.641} C_VEL
LIN {X 0,Y 258.742,Z 406.011,A -85,B 0,C 180,E1 -18508.931,E2 -18508.931} C_VEL
LIN {X 0,Y 257.126,Z 402.111,A -85,B 0,C 180,E1 -18511,E2 -18511} C_VEL
LIN {X 0,Y 256.074,Z 399.207,A -85,B 0,C 180,E1 -18512.632,E2 -18512.632} C_VEL
LIN {X 0,Y 256.074,Z 399.207,A -85,B 0,C 180,E1 -18515.69,E2 -18515.69} C_VEL
LIN {X 0,Y 256.11,Z 399.202,A -85,B 0,C 180,E1 -18519.1,E2 -18519.1} C_VEL
LIN {X 0,Y 256.203,Z 399.199,A -85,B 0,C 180,E1 -18524.079,E2 -18524.079} C_VEL
LIN {X 0,Y 256.262,Z 399.184,A -85,B 0,C 180,E1 -18528.932,E2 -18528.932} C_VEL
LIN {X 0,Y 256.478,Z 399.162,A -85,B 0,C 180,E1 -18532.126,E2 -18532.126} C_VEL
LIN {X 0,Y 256.442,Z 399.157,A -85,B 0,C 180,E1 -18536.858,E2 -18536.858} C_VEL
LIN {X 0,Y 256.686,Z 399.129,A -85,B 0,C 180,E1 -18538.431,E2 -18538.431} C_VEL
LIN {X 0,Y 256.69,Z 399.125,A -85,B 0,C 180,E1 -18541.569,E2 -18541.569} C_VEL
LIN {X 0,Y 256.425,Z 399.122,A -85,B 0,C 180,E1 -18546.754,E2 -18546.754} C_VEL
LIN {X 0,Y 256.391,Z 399.155,A -85,B 0,C 180,E1 -18549.467,E2 -18549.467} C_VEL
LIN {X 0,Y 256.226,Z 399.154,A -85,B 0,C 180,E1 -18554.292,E2 -18554.292} C_VEL
LIN {X 0,Y 256.169,Z 399.201,A -85,B 0,C 180,E1 -18557.565,E2 -18557.565} C_VEL
LIN {X 0,Y 256.129,Z 399.171,A -85,B 0,C 180,E1 -18561.109,E2 -18561.109} C_VEL
LIN {X 0,Y 256.076,Z 399.198,A -85,B 0,C 180,E1 -18565.089,E2 -18565.089} C_VEL
LIN {X 0,Y 256.06,Z 399.195,A -85,B 0,C 180,E1 -18567.204,E2 -18567.204} C_VEL
LIN {X 0,Y 256.826,Z 401.622,A -85,B 0,C 180,E1 -18567.613,E2 -18567.613} C_VEL
LIN {X 0,Y 258.888,Z 404.02,A -85,B 0,C 180,E1 -18568.469,E2 -18568.469} C_VEL
LIN {X 0,Y 260.303,Z 405.098,A -85,B 0,C 180,E1 -18569.009,E2 -18569.009} C_VEL
LIN {X 0,Y 262.399,Z 408.446,A -85,B 0,C 180,E1 -18569.869,E2 -18569.869} C_VEL
LIN {X 0,Y 264.503,Z 410.51,A -85,B 0,C 180,E1 -18570.639,E2 -18570.639} C_VEL
LIN {X 0,Y 266.976,Z 413.957,A -85,B 0,C 180,E1 -18571.556,E2 -18571.556} C_VEL
LIN {X 0,Y 268.419,Z 415.691,A -85,B 0,C 180,E1 -18572.061,E2 -18572.061} C_VEL
LIN {X 0,Y 272.587,Z 421.287,A -85,B 0,C 180,E1 -18573.482,E2 -18573.482} C_VEL
LIN {X 0,Y 275.609,Z 425.33,A -85,B 0,C 180,E1 -18574.457,E2 -18574.457} C_VEL
LIN {X 0,Y 283.354,Z 436.593,A -85,B 0,C 180,E1 -18576.809,E2 -18576.809} C_VEL
LIN {X 0,Y 291.919,Z 450.181,A -85,B 0,C 180,E1 -18579.186,E2 -18579.186} C_VEL
LIN {X 0,Y 298.735,Z 462.325,A -85,B 0,C 180,E1 -18580.955,E2 -18580.955} C_VEL
LIN {X 0,Y 296.271,Z 510.82,A -85,B 0,C 180,E1 -18582.098,E2 -18582.098} C_VEL
LIN {X 0,Y 295.324,Z 536.581,A -85,B 0,C 180,E1 -18582.842,E2 -18582.842} C_VEL
LIN {X 0,Y 294.201,Z 551.244,A -85,B 0,C 180,E1 -18583.508,E2 -18583.508} C_VEL
LIN {X 0,Y 292.559,Z 564.791,A -85,B 0,C 180,E1 -18584.345,E2 -18584.345} C_VEL
LIN {X 0,Y 290.458,Z 578.236,A -85,B 0,C 180,E1 -18585.439,E2 -18585.439} C_VEL
LIN {X 0,Y 287.714,Z 592.043,A -85,B 0,C 180,E1 -18586.848,E2 -18586.848} C_VEL
LIN {X 0,Y 284.291,Z 605.895,A -85,B 0,C 180,E1 -18588.604,E2 -18588.604} C_VEL
LIN {X 0,Y 280.734,Z 618.265,A -85,B 0,C 180,E1 -18590.564,E2 -18590.564} C_VEL
LIN {X 0,Y 277.414,Z 628.535,A -85,B 0,C 180,E1 -18592.556,E2 -18592.556} C_VEL
LIN {X 0,Y 273.904,Z 638.268,A -85,B 0,C 180,E1 -18594.83,E2 -18594.83} C_VEL
LIN {X 0,Y 270.47,Z 647.149,A -85,B 0,C 180,E1 -18597.374,E2 -18597.374} C_VEL
LIN {X 0,Y 267.273,Z 654.697,A -85,B 0,C 180,E1 -18600.027,E2 -18600.027} C_VEL
LIN {X 0,Y 264.193,Z 661.661,A -85,B 0,C 180,E1 -18603.115,E2 -18603.115} C_VEL
LIN {X 0,Y 261.707,Z 667.064,A -85,B 0,C 180,E1 -18606.247,E2 -18606.247} C_VEL
LIN {X 0,Y 259.702,Z 671.086,A -85,B 0,C 180,E1 -18609.404,E2 -18609.404} C_VEL
LIN {X 0,Y 258.254,Z 673.846,A -85,B 0,C 180,E1 -18612.583,E2 -18612.583} C_VEL
LIN {X 0,Y 257.238,Z 675.44,A -85,B 0,C 180,E1 -18615.767,E2 -18615.767} C_VEL
LIN {X 0,Y 256.779,Z 675.888,A -85,B 0,C 180,E1 -18618.955,E2 -18618.955} C_VEL
LIN {X 0,Y 256.65,Z 675.192,A -85,B 0,C 180,E1 -18622.131,E2 -18622.131} C_VEL
LIN {X 0,Y 256.704,Z 673.428,A -85,B 0,C 180,E1 -18625.29,E2 -18625.29} C_VEL
LIN {X 0,Y 257.262,Z 670.52,A -85,B 0,C 180,E1 -18628.435,E2 -18628.435} C_VEL
LIN {X 0,Y 258.244,Z 666.419,A -85,B 0,C 180,E1 -18631.56,E2 -18631.56} C_VEL
LIN {X 0,Y 259.62,Z 661.04,A -85,B 0,C 180,E1 -18634.659,E2 -18634.659} C_VEL
LIN {X 0,Y 261.453,Z 654.224,A -85,B 0,C 180,E1 -18637.724,E2 -18637.724} C_VEL
LIN {X 0,Y 263.365,Z 646.958,A -85,B 0,C 180,E1 -18640.377,E2 -18640.377} C_VEL
LIN {X 0,Y 265.721,Z 638.182,A -85,B 0,C 180,E1 -18642.992,E2 -18642.992} C_VEL
LIN {X 0,Y 268.378,Z 627.645,A -85,B 0,C 180,E1 -18645.57,E2 -18645.57} C_VEL
LIN {X 0,Y 271.086,Z 615.815,A -85,B 0,C 180,E1 -18647.931,E2 -18647.931} C_VEL
LIN {X 0,Y 273.464,Z 603.812,A -85,B 0,C 180,E1 -18649.909,E2 -18649.909} C_VEL
LIN {X 0,Y 276.042,Z 590.482,A -85,B 0,C 180,E1 -18651.664,E2 -18651.664} C_VEL
LIN {X 0,Y 278.074,Z 577.46,A -85,B 0,C 180,E1 -18653.063,E2 -18653.063} C_VEL
LIN {X 0,Y 279.905,Z 563.072,A -85,B 0,C 180,E1 -18654.277,E2 -18654.277} C_VEL
LIN {X 0,Y 281.355,Z 547.676,A -85,B 0,C 180,E1 -18655.251,E2 -18655.251} C_VEL
LIN {X 0,Y 282.131,Z 532.628,A -85,B 0,C 180,E1 -18655.932,E2 -18655.932} C_VEL
LIN {X 0,Y 283.386,Z 492.126,A -85,B 0,C 180,E1 -18657.015,E2 -18657.015} C_VEL
LIN {X 0,Y 284.944,Z 450.766,A -85,B 0,C 180,E1 -18658.043,E2 -18658.043} C_VEL
LIN {X 0,Y 276.092,Z 433.14,A -85,B 0,C 180,E1 -18659.868,E2 -18659.868} C_VEL
LIN {X 0,Y 267.244,Z 417.688,A -85,B 0,C 180,E1 -18661.786,E2 -18661.786} C_VEL
LIN {X 0,Y 260.38,Z 406.855,A -85,B 0,C 180,E1 -18663.357,E2 -18663.357} C_VEL
LIN {X 0,Y 258.327,Z 403.521,A -85,B 0,C 180,E1 -18663.854,E2 -18663.854} C_VEL
LIN {X 0,Y 256.643,Z 401.116,A -85,B 0,C 180,E1 -18664.258,E2 -18664.258} C_VEL
LIN {X 0,Y 256.111,Z 399.205,A -85,B 0,C 180,E1 -18664.481,E2 -18664.481} C_VEL
LIN {X 0,Y 256.116,Z 399.202,A -85,B 0,C 180,E1 -18667.27,E2 -18667.27} C_VEL
LIN {X 0,Y 256.027,Z 399.218,A -85,B 0,C 180,E1 -18672.169,E2 -18672.169} C_VEL
LIN {X 0,Y 256.02,Z 399.214,A -85,B 0,C 180,E1 -18676.663,E2 -18676.663} C_VEL
LIN {X 0,Y 256.041,Z 399.212,A -85,B 0,C 180,E1 -18680.852,E2 -18680.852} C_VEL
LIN {X 0,Y 256.076,Z 399.212,A -85,B 0,C 180,E1 -18684.806,E2 -18684.806} C_VEL
LIN {X 0,Y 256.075,Z 399.214,A -85,B 0,C 180,E1 -18688.569,E2 -18688.569} C_VEL
LIN {X 0,Y 256.076,Z 399.209,A -85,B 0,C 180,E1 -18692.188,E2 -18692.188} C_VEL
LIN {X 0,Y 256.129,Z 399.194,A -85,B 0,C 180,E1 -18695.695,E2 -18695.695} C_VEL
LIN {X 0,Y 256.121,Z 399.207,A -85,B 0,C 180,E1 -18699.101,E2 -18699.101} C_VEL
LIN {X 0,Y 256.227,Z 399.193,A -85,B 0,C 180,E1 -18704.08,E2 -18704.08} C_VEL
LIN {X 0,Y 256.274,Z 399.128,A -85,B 0,C 180,E1 -18708.932,E2 -18708.932} C_VEL
LIN {X 0,Y 256.396,Z 399.122,A -85,B 0,C 180,E1 -18710.609,E2 -18710.609} C_VEL
LIN {X 0,Y 255.723,Z 399.228,A -85,B 0,C 180,E1 -18711.92,E2 -18711.92} C_VEL
LIN {X 0,Y 252.798,Z 399.621,A -85,B 0,C 180,E1 -18714.055,E2 -18714.055} C_VEL
LIN {X 0,Y 250.393,Z 399.915,A -85,B 0,C 180,E1 -18715.793,E2 -18715.793} C_VEL
LIN {X 0,Y 249.484,Z 400.017,A -85,B 0,C 180,E1 -18717.143,E2 -18717.143} C_VEL
LIN {X 0,Y 249.476,Z 400.016,A -85,B 0,C 180,E1 -18717.599,E2 -18717.599} C_VEL
LIN {X 0,Y 249.657,Z 400.009,A -85,B 0,C 180,E1 -18720,E2 -18720} C_VEL
LIN {X 0,Y 249.651,Z 400.009,A -85,B 0,C 180,E1 -18721.613,E2 -18721.613} C_VEL
LIN {X 0,Y 249.418,Z 400.04,A -85,B 0,C 180,E1 -18726.471,E2 -18726.471} C_VEL
LIN {X 0,Y 249.328,Z 400.038,A -85,B 0,C 180,E1 -18729.737,E2 -18729.737} C_VEL
LIN {X 0,Y 249.138,Z 400.064,A -85,B 0,C 180,E1 -18734.707,E2 -18734.707} C_VEL
LIN {X 0,Y 249.071,Z 400.078,A -85,B 0,C 180,E1 -18738.082,E2 -18738.082} C_VEL
LIN {X 0,Y 249.039,Z 400.088,A -85,B 0,C 180,E1 -18741.522,E2 -18741.522} C_VEL
LIN {X 0,Y 249.04,Z 400.086,A -85,B 0,C 180,E1 -18745.44,E2 -18745.44} C_VEL
LIN {X 0,Y 249.02,Z 400.088,A -85,B 0,C 180,E1 -18748.968,E2 -18748.968} C_VEL
LIN {X 0,Y 249.022,Z 400.079,A -85,B 0,C 180,E1 -18752.427,E2 -18752.427} C_VEL
LIN {X 0,Y 249.053,Z 400.167,A -85,B 0,C 180,E1 -18756.754,E2 -18756.754} C_VEL
LIN {X 0,Y 252.954,Z 411.904,A -85,B 0,C 180,E1 -18760.842,E2 -18760.842} C_VEL
LIN {X 0,Y 256.257,Z 422.799,A -85,B 0,C 180,E1 -18764.285,E2 -18764.285} C_VEL
LIN {X 0,Y 257.777,Z 428.149,A -85,B 0,C 180,E1 -18765.838,E2 -18765.838} C_VEL
LIN {X 0,Y 265.675,Z 445.068,A -85,B 0,C 180,E1 -18767.79,E2 -18767.79} C_VEL
LIN {X 0,Y 271.046,Z 457.848,A -85,B 0,C 180,E1 -18769.069,E2 -18769.069} C_VEL
LIN {X 0,Y 274.318,Z 488.592,A -85,B 0,C 180,E1 -18770.536,E2 -18770.536} C_VEL
LIN {X 0,Y 277.177,Z 519.193,A -85,B 0,C 180,E1 -18771.884,E2 -18771.884} C_VEL
LIN {X 0,Y 273.747,Z 599.909,A -85,B 0,C 180,E1 -18773.923,E2 -18773.923} C_VEL
LIN {X 0,Y 272.359,Z 615.486,A -85,B 0,C 180,E1 -18774.565,E2 -18774.565} C_VEL
LIN {X 0,Y 270.368,Z 630.542,A -85,B 0,C 180,E1 -18775.459,E2 -18775.459} C_VEL
LIN {X 0,Y 267.938,Z 644.651,A -85,B 0,C 180,E1 -18776.576,E2 -18776.576} C_VEL
LIN {X 0,Y 265.322,Z 656.831,A -85,B 0,C 180,E1 -18777.786,E2 -18777.786} C_VEL
LIN {X 0,Y 262.712,Z 668.326,A -85,B 0,C 180,E1 -18779.19,E2 -18779.19} C_VEL
LIN {X 0,Y 259.856,Z 680.92,A -85,B 0,C 180,E1 -18781.09,E2 -18781.09} C_VEL
LIN {X 0,Y 256.889,Z 692.334,A -85,B 0,C 180,E1 -18783.166,E2 -18783.166} C_VEL
LIN {X 0,Y 254.257,Z 702.901,A -85,B 0,C 180,E1 -18785.505,E2 -18785.505} C_VEL
LIN {X 0,Y 251.814,Z 713.264,A -85,B 0,C 180,E1 -18788.297,E2 -18788.297} C_VEL
LIN {X 0,Y 249.995,Z 721.908,A -85,B 0,C 180,E1 -18791.138,E2 -18791.138} C_VEL
LIN {X 0,Y 248.851,Z 728.568,A -85,B 0,C 180,E1 -18793.784,E2 -18793.784} C_VEL
LIN {X 0,Y 248.132,Z 735.038,A -85,B 0,C 180,E1 -18796.903,E2 -18796.903} C_VEL
LIN {X 0,Y 248.046,Z 740.451,A -85,B 0,C 180,E1 -18800.212,E2 -18800.212} C_VEL
LIN {X 0,Y 248.395,Z 744.476,A -85,B 0,C 180,E1 -18803.501,E2 -18803.501} C_VEL
LIN {X 0,Y 248.679,Z 745.99,A -85,B 0,C 180,E1 -18805.136,E2 -18805.136} C_VEL
LIN {X 0,Y 249.179,Z 748.005,A -85,B 0,C 180,E1 -18808.383,E2 -18808.383} C_VEL
